   // UNI[3596] := 16#6DAE;
   // UNI[3597] := 16#6DAF;
   // UNI[3598] := 16#6DB2;
   // UNI[3599] := 16#6DB5;
   // UNI[3600] := 16#6DB8;
   // UNI[3601] := 16#6DBF;
   // UNI[3602] := 16#6DC0;
   // UNI[3603] := 16#6DC4;
   // UNI[3604] := 16#6DC5;
   // UNI[3605] := 16#6DC6;
   // UNI[3606] := 16#6DC7;
   // UNI[3607] := 16#6DCB;
   // UNI[3608] := 16#6DCC;
   // UNI[3609] := 16#6DD1;
   // UNI[3610] := 16#6DD6;
   // UNI[3611] := 16#6DD8;
   // UNI[3612] := 16#6DD9;
   // UNI[3613] := 16#6DDD;
   // UNI[3614] := 16#6DDE;
   // UNI[3615] := 16#6DE0;
   // UNI[3616] := 16#6DE1;
   // UNI[3617] := 16#6DE4;
   // UNI[3618] := 16#6DE6;
   // UNI[3619] := 16#6DEB;
   // UNI[3620] := 16#6DEC;
   // UNI[3621] := 16#6DEE;
   // UNI[3622] := 16#6DF1;
   // UNI[3623] := 16#6DF3;
   // UNI[3624] := 16#6DF7;
   // UNI[3625] := 16#6DF9;
   // UNI[3626] := 16#6DFB;
   // UNI[3627] := 16#6DFC;
   // UNI[3628] := 16#6E05;
   // UNI[3629] := 16#6E0A;
   // UNI[3630] := 16#6E0C;
   // UNI[3631] := 16#6E0D;
   // UNI[3632] := 16#6E0E;
   // UNI[3633] := 16#6E10;
   // UNI[3634] := 16#6E11;
   // UNI[3635] := 16#6E14;
   // UNI[3636] := 16#6E16;
   // UNI[3637] := 16#6E17;
   // UNI[3638] := 16#6E1A;
   // UNI[3639] := 16#6E1D;
   // UNI[3640] := 16#6E20;
   // UNI[3641] := 16#6E21;
   // UNI[3642] := 16#6E23;
   // UNI[3643] := 16#6E24;
   // UNI[3644] := 16#6E25;
   // UNI[3645] := 16#6E29;
   // UNI[3646] := 16#6E2B;
   // UNI[3647] := 16#6E2D;
   // UNI[3648] := 16#6E2F;
   // UNI[3649] := 16#6E32;
   // UNI[3650] := 16#6E34;
   // UNI[3651] := 16#6E38;
   // UNI[3652] := 16#6E3A;
   // UNI[3653] := 16#6E43;
   // UNI[3654] := 16#6E44;
   // UNI[3655] := 16#6E4D;
   // UNI[3656] := 16#6E4E;
   // UNI[3657] := 16#6E53;
   // UNI[3658] := 16#6E54;
   // UNI[3659] := 16#6E56;
   // UNI[3660] := 16#6E58;
   // UNI[3661] := 16#6E5B;
   // UNI[3662] := 16#6E5F;
   // UNI[3663] := 16#6E6B;
   // UNI[3664] := 16#6E6E;
   // UNI[3665] := 16#6E7E;
   // UNI[3666] := 16#6E7F;
   // UNI[3667] := 16#6E83;
   // UNI[3668] := 16#6E85;
   // UNI[3669] := 16#6E86;
   // UNI[3670] := 16#6E89;
   // UNI[3671] := 16#6E8F;
   // UNI[3672] := 16#6E90;
   // UNI[3673] := 16#6E98;
   // UNI[3674] := 16#6E9C;
   // UNI[3675] := 16#6E9F;
   // UNI[3676] := 16#6EA2;
   // UNI[3677] := 16#6EA5;
   // UNI[3678] := 16#6EA7;
   // UNI[3679] := 16#6EAA;
   // UNI[3680] := 16#6EAF;
   // UNI[3681] := 16#6EB1;
   // UNI[3682] := 16#6EB2;
   // UNI[3683] := 16#6EB4;
   // UNI[3684] := 16#6EB6;
   // UNI[3685] := 16#6EB7;
   // UNI[3686] := 16#6EBA;
   // UNI[3687] := 16#6EBB;
   // UNI[3688] := 16#6EBD;
   // UNI[3689] := 16#6EC1;
   // UNI[3690] := 16#6EC2;
   // UNI[3691] := 16#6EC7;
   // UNI[3692] := 16#6ECB;
   // UNI[3693] := 16#6ECF;
   // UNI[3694] := 16#6ED1;
   // UNI[3695] := 16#6ED3;
   // UNI[3696] := 16#6ED4;
   // UNI[3697] := 16#6ED5;
   // UNI[3698] := 16#6ED7;
   // UNI[3699] := 16#6EDA;
   // UNI[3700] := 16#6EDE;
   // UNI[3701] := 16#6EDF;
   // UNI[3702] := 16#6EE0;
   // UNI[3703] := 16#6EE1;
   // UNI[3704] := 16#6EE2;
   // UNI[3705] := 16#6EE4;
   // UNI[3706] := 16#6EE5;
   // UNI[3707] := 16#6EE6;
   // UNI[3708] := 16#6EE8;
   // UNI[3709] := 16#6EE9;
   // UNI[3710] := 16#6EF4;
   // UNI[3711] := 16#6EF9;
   // UNI[3712] := 16#6F02;
   // UNI[3713] := 16#6F06;
   // UNI[3714] := 16#6F09;
   // UNI[3715] := 16#6F0F;
   // UNI[3716] := 16#6F13;
   // UNI[3717] := 16#6F14;
   // UNI[3718] := 16#6F15;
   // UNI[3719] := 16#6F20;
   // UNI[3720] := 16#6F24;
   // UNI[3721] := 16#6F29;
   // UNI[3722] := 16#6F2A;
   // UNI[3723] := 16#6F2B;
   // UNI[3724] := 16#6F2D;
   // UNI[3725] := 16#6F2F;
   // UNI[3726] := 16#6F31;
   // UNI[3727] := 16#6F33;
   // UNI[3728] := 16#6F36;
   // UNI[3729] := 16#6F3E;
   // UNI[3730] := 16#6F46;
   // UNI[3731] := 16#6F47;
   // UNI[3732] := 16#6F4B;
   // UNI[3733] := 16#6F4D;
   // UNI[3734] := 16#6F58;
   // UNI[3735] := 16#6F5C;
   // UNI[3736] := 16#6F5E;
   // UNI[3737] := 16#6F62;
   // UNI[3738] := 16#6F66;
   // UNI[3739] := 16#6F6D;
   // UNI[3740] := 16#6F6E;
   // UNI[3741] := 16#6F72;
   // UNI[3742] := 16#6F74;
   // UNI[3743] := 16#6F78;
   // UNI[3744] := 16#6F7A;
   // UNI[3745] := 16#6F7C;
   // UNI[3746] := 16#6F84;
   // UNI[3747] := 16#6F88;
   // UNI[3748] := 16#6F89;
   // UNI[3749] := 16#6F8C;
   // UNI[3750] := 16#6F8D;
   // UNI[3751] := 16#6F8E;
   // UNI[3752] := 16#6F9C;
   // UNI[3753] := 16#6FA1;
   // UNI[3754] := 16#6FA7;
   // UNI[3755] := 16#6FB3;
   // UNI[3756] := 16#6FB6;
   // UNI[3757] := 16#6FB9;
   // UNI[3758] := 16#6FC0;
   // UNI[3759] := 16#6FC2;
   // UNI[3760] := 16#6FC9;
   // UNI[3761] := 16#6FD1;
   // UNI[3762] := 16#6FD2;
   // UNI[3763] := 16#6FDE;
   // UNI[3764] := 16#6FE0;
   // UNI[3765] := 16#6FE1;
   // UNI[3766] := 16#6FEE;
   // UNI[3767] := 16#6FEF;
   // UNI[3768] := 16#7011;
   // UNI[3769] := 16#701A;
   // UNI[3770] := 16#701B;
   // UNI[3771] := 16#7023;
   // UNI[3772] := 16#7035;
   // UNI[3773] := 16#7039;
   // UNI[3774] := 16#704C;
   // UNI[3775] := 16#704F;
   // UNI[3776] := 16#705E;
   // UNI[3777] := 16#706B;
   // UNI[3778] := 16#706C;
   // UNI[3779] := 16#706D;
   // UNI[3780] := 16#706F;
   // UNI[3781] := 16#7070;
   // UNI[3782] := 16#7075;
   // UNI[3783] := 16#7076;
   // UNI[3784] := 16#7078;
   // UNI[3785] := 16#707C;
   // UNI[3786] := 16#707E;
   // UNI[3787] := 16#707F;
   // UNI[3788] := 16#7080;
   // UNI[3789] := 16#7085;
   // UNI[3790] := 16#7089;
   // UNI[3791] := 16#708A;
   // UNI[3792] := 16#708E;
   // UNI[3793] := 16#7092;
   // UNI[3794] := 16#7094;
   // UNI[3795] := 16#7095;
   // UNI[3796] := 16#7096;
   // UNI[3797] := 16#7099;
   // UNI[3798] := 16#709C;
   // UNI[3799] := 16#709D;
   // UNI[3800] := 16#70AB;
   // UNI[3801] := 16#70AC;
   // UNI[3802] := 16#70AD;
   // UNI[3803] := 16#70AE;
   // UNI[3804] := 16#70AF;
   // UNI[3805] := 16#70B1;
   // UNI[3806] := 16#70B3;
   // UNI[3807] := 16#70B7;
   // UNI[3808] := 16#70B8;
   // UNI[3809] := 16#70B9;
   // UNI[3810] := 16#70BB;
   // UNI[3811] := 16#70BC;
   // UNI[3812] := 16#70BD;
   // UNI[3813] := 16#70C0;
   // UNI[3814] := 16#70C1;
   // UNI[3815] := 16#70C2;
   // UNI[3816] := 16#70C3;
   // UNI[3817] := 16#70C8;
   // UNI[3818] := 16#70CA;
   // UNI[3819] := 16#70D8;
   // UNI[3820] := 16#70D9;
   // UNI[3821] := 16#70DB;
   // UNI[3822] := 16#70DF;
   // UNI[3823] := 16#70E4;
   // UNI[3824] := 16#70E6;
   // UNI[3825] := 16#70E7;
   // UNI[3826] := 16#70E8;
   // UNI[3827] := 16#70E9;
   // UNI[3828] := 16#70EB;
   // UNI[3829] := 16#70EC;
   // UNI[3830] := 16#70ED;
   // UNI[3831] := 16#70EF;
   // UNI[3832] := 16#70F7;
   // UNI[3833] := 16#70F9;
   // UNI[3834] := 16#70FD;
   // UNI[3835] := 16#7109;
   // UNI[3836] := 16#710A;
   // UNI[3837] := 16#7110;
   // UNI[3838] := 16#7113;
   // UNI[3839] := 16#7115;
   // UNI[3840] := 16#7116;
   // UNI[3841] := 16#7118;
   // UNI[3842] := 16#7119;
   // UNI[3843] := 16#711A;
   // UNI[3844] := 16#7126;
   // UNI[3845] := 16#712F;
   // UNI[3846] := 16#7130;
   // UNI[3847] := 16#7131;
   // UNI[3848] := 16#7136;
   // UNI[3849] := 16#7145;
   // UNI[3850] := 16#714A;
   // UNI[3851] := 16#714C;
   // UNI[3852] := 16#714E;
   // UNI[3853] := 16#715C;
   // UNI[3854] := 16#715E;
   // UNI[3855] := 16#7164;
   // UNI[3856] := 16#7166;
   // UNI[3857] := 16#7167;
   // UNI[3858] := 16#7168;
   // UNI[3859] := 16#716E;
   // UNI[3860] := 16#7172;
   // UNI[3861] := 16#7173;
   // UNI[3862] := 16#7178;
   // UNI[3863] := 16#717A;
   // UNI[3864] := 16#717D;
   // UNI[3865] := 16#7184;
   // UNI[3866] := 16#718A;
   // UNI[3867] := 16#718F;
   // UNI[3868] := 16#7194;
   // UNI[3869] := 16#7198;
   // UNI[3870] := 16#7199;
   // UNI[3871] := 16#719F;
   // UNI[3872] := 16#71A0;
   // UNI[3873] := 16#71A8;
   // UNI[3874] := 16#71AC;
   // UNI[3875] := 16#71B3;
   // UNI[3876] := 16#71B5;
   // UNI[3877] := 16#71B9;
   // UNI[3878] := 16#71C3;
   // UNI[3879] := 16#71CE;
   // UNI[3880] := 16#71D4;
   // UNI[3881] := 16#71D5;
   // UNI[3882] := 16#71E0;
   // UNI[3883] := 16#71E5;
   // UNI[3884] := 16#71E7;
   // UNI[3885] := 16#71EE;
   // UNI[3886] := 16#71F9;
   // UNI[3887] := 16#7206;
   // UNI[3888] := 16#721D;
   // UNI[3889] := 16#7228;
   // UNI[3890] := 16#722A;
   // UNI[3891] := 16#722C;
   // UNI[3892] := 16#7230;
   // UNI[3893] := 16#7231;
   // UNI[3894] := 16#7235;
   // UNI[3895] := 16#7236;
   // UNI[3896] := 16#7237;
   // UNI[3897] := 16#7238;
   // UNI[3898] := 16#7239;
   // UNI[3899] := 16#723B;
   // UNI[3900] := 16#723D;
   // UNI[3901] := 16#723F;
   // UNI[3902] := 16#7247;
   // UNI[3903] := 16#7248;
   // UNI[3904] := 16#724C;
   // UNI[3905] := 16#724D;
   // UNI[3906] := 16#7252;
   // UNI[3907] := 16#7256;
   // UNI[3908] := 16#7259;
   // UNI[3909] := 16#725B;
   // UNI[3910] := 16#725D;
   // UNI[3911] := 16#725F;
   // UNI[3912] := 16#7261;
   // UNI[3913] := 16#7262;
   // UNI[3914] := 16#7266;
   // UNI[3915] := 16#7267;
   // UNI[3916] := 16#7269;
   // UNI[3917] := 16#726E;
   // UNI[3918] := 16#726F;
   // UNI[3919] := 16#7272;
   // UNI[3920] := 16#7275;
   // UNI[3921] := 16#7279;
   // UNI[3922] := 16#727A;
   // UNI[3923] := 16#727E;
   // UNI[3924] := 16#727F;
   // UNI[3925] := 16#7280;
   // UNI[3926] := 16#7281;
   // UNI[3927] := 16#7284;
   // UNI[3928] := 16#728A;
   // UNI[3929] := 16#728B;
   // UNI[3930] := 16#728D;
   // UNI[3931] := 16#728F;
   // UNI[3932] := 16#7292;
   // UNI[3933] := 16#729F;
   // UNI[3934] := 16#72AC;
   // UNI[3935] := 16#72AD;
   // UNI[3936] := 16#72AF;
   // UNI[3937] := 16#72B0;
   // UNI[3938] := 16#72B4;
   // UNI[3939] := 16#72B6;
   // UNI[3940] := 16#72B7;
   // UNI[3941] := 16#72B8;
   // UNI[3942] := 16#72B9;
   // UNI[3943] := 16#72C1;
   // UNI[3944] := 16#72C2;
   // UNI[3945] := 16#72C3;
   // UNI[3946] := 16#72C4;
   // UNI[3947] := 16#72C8;
   // UNI[3948] := 16#72CD;
   // UNI[3949] := 16#72CE;
   // UNI[3950] := 16#72D0;
   // UNI[3951] := 16#72D2;
   // UNI[3952] := 16#72D7;
   // UNI[3953] := 16#72D9;
   // UNI[3954] := 16#72DE;
   // UNI[3955] := 16#72E0;
   // UNI[3956] := 16#72E1;
   // UNI[3957] := 16#72E8;
   // UNI[3958] := 16#72E9;
   // UNI[3959] := 16#72EC;
   // UNI[3960] := 16#72ED;
   // UNI[3961] := 16#72EE;
   // UNI[3962] := 16#72EF;
   // UNI[3963] := 16#72F0;
   // UNI[3964] := 16#72F1;
   // UNI[3965] := 16#72F2;
   // UNI[3966] := 16#72F3;
   // UNI[3967] := 16#72F4;
   // UNI[3968] := 16#72F7;
   // UNI[3969] := 16#72F8;
   // UNI[3970] := 16#72FA;
   // UNI[3971] := 16#72FB;
   // UNI[3972] := 16#72FC;
   // UNI[3973] := 16#7301;
   // UNI[3974] := 16#7303;
   // UNI[3975] := 16#730A;
   // UNI[3976] := 16#730E;
   // UNI[3977] := 16#7313;
   // UNI[3978] := 16#7315;
   // UNI[3979] := 16#7316;
   // UNI[3980] := 16#7317;
   // UNI[3981] := 16#731B;
   // UNI[3982] := 16#731C;
   // UNI[3983] := 16#731D;
   // UNI[3984] := 16#731E;
   // UNI[3985] := 16#7321;
   // UNI[3986] := 16#7322;
   // UNI[3987] := 16#7325;
   // UNI[3988] := 16#7329;
   // UNI[3989] := 16#732A;
   // UNI[3990] := 16#732B;
   // UNI[3991] := 16#732C;
   // UNI[3992] := 16#732E;
   // UNI[3993] := 16#7331;
   // UNI[3994] := 16#7334;
   // UNI[3995] := 16#7337;
   // UNI[3996] := 16#7338;
   // UNI[3997] := 16#7339;
   // UNI[3998] := 16#733E;
   // UNI[3999] := 16#733F;
   // UNI[4000] := 16#734D;
   // UNI[4001] := 16#7350;
   // UNI[4002] := 16#7352;
   // UNI[4003] := 16#7357;
   // UNI[4004] := 16#7360;
   // UNI[4005] := 16#736C;
   // UNI[4006] := 16#736D;
   // UNI[4007] := 16#736F;
   // UNI[4008] := 16#737E;
   // UNI[4009] := 16#7384;
   // UNI[4010] := 16#7387;
   // UNI[4011] := 16#7389;
   // UNI[4012] := 16#738B;
   // UNI[4013] := 16#738E;
   // UNI[4014] := 16#7391;
   // UNI[4015] := 16#7396;
   // UNI[4016] := 16#739B;
   // UNI[4017] := 16#739F;
   // UNI[4018] := 16#73A2;
   // UNI[4019] := 16#73A9;
   // UNI[4020] := 16#73AB;
   // UNI[4021] := 16#73AE;
   // UNI[4022] := 16#73AF;
   // UNI[4023] := 16#73B0;
   // UNI[4024] := 16#73B2;
   // UNI[4025] := 16#73B3;
   // UNI[4026] := 16#73B7;
   // UNI[4027] := 16#73BA;
   // UNI[4028] := 16#73BB;
   // UNI[4029] := 16#73C0;
   // UNI[4030] := 16#73C2;
   // UNI[4031] := 16#73C8;
   // UNI[4032] := 16#73C9;
   // UNI[4033] := 16#73CA;
   // UNI[4034] := 16#73CD;
   // UNI[4035] := 16#73CF;
   // UNI[4036] := 16#73D0;
   // UNI[4037] := 16#73D1;
   // UNI[4038] := 16#73D9;
   // UNI[4039] := 16#73DE;
   // UNI[4040] := 16#73E0;
   // UNI[4041] := 16#73E5;
   // UNI[4042] := 16#73E7;
   // UNI[4043] := 16#73E9;
   // UNI[4044] := 16#73ED;
   // UNI[4045] := 16#73F2;
   // UNI[4046] := 16#7403;
   // UNI[4047] := 16#7405;
   // UNI[4048] := 16#7406;
   // UNI[4049] := 16#7409;
   // UNI[4050] := 16#740A;
   // UNI[4051] := 16#740F;
   // UNI[4052] := 16#7410;
   // UNI[4053] := 16#741A;
   // UNI[4054] := 16#741B;
   // UNI[4055] := 16#7422;
   // UNI[4056] := 16#7425;
   // UNI[4057] := 16#7426;
   // UNI[4058] := 16#7428;
   // UNI[4059] := 16#742A;
   // UNI[4060] := 16#742C;
   // UNI[4061] := 16#742E;
   // UNI[4062] := 16#7430;
   // UNI[4063] := 16#7433;
   // UNI[4064] := 16#7434;
   // UNI[4065] := 16#7435;
   // UNI[4066] := 16#7436;
   // UNI[4067] := 16#743C;
   // UNI[4068] := 16#7441;
   // UNI[4069] := 16#7455;
   // UNI[4070] := 16#7457;
   // UNI[4071] := 16#7459;
   // UNI[4072] := 16#745A;
   // UNI[4073] := 16#745B;
   // UNI[4074] := 16#745C;
   // UNI[4075] := 16#745E;
   // UNI[4076] := 16#745F;
   // UNI[4077] := 16#746D;
   // UNI[4078] := 16#7470;
   // UNI[4079] := 16#7476;
   // UNI[4080] := 16#7477;
   // UNI[4081] := 16#747E;
   // UNI[4082] := 16#7480;
   // UNI[4083] := 16#7481;
   // UNI[4084] := 16#7483;
   // UNI[4085] := 16#7487;
   // UNI[4086] := 16#748B;
   // UNI[4087] := 16#748E;
   // UNI[4088] := 16#7490;
   // UNI[4089] := 16#749C;
   // UNI[4090] := 16#749E;
   // UNI[4091] := 16#74A7;
   // UNI[4092] := 16#74A8;
   // UNI[4093] := 16#74A9;
   // UNI[4094] := 16#74BA;
   // UNI[4095] := 16#74D2;
   // UNI[4096] := 16#74DC;
   // UNI[4097] := 16#74DE;
   // UNI[4098] := 16#74E0;
   // UNI[4099] := 16#74E2;
   // UNI[4100] := 16#74E3;
   // UNI[4101] := 16#74E4;
   // UNI[4102] := 16#74E6;
   // UNI[4103] := 16#74EE;
   // UNI[4104] := 16#74EF;
   // UNI[4105] := 16#74F4;
   // UNI[4106] := 16#74F6;
   // UNI[4107] := 16#74F7;
   // UNI[4108] := 16#74FF;
   // UNI[4109] := 16#7504;
   // UNI[4110] := 16#750D;
   // UNI[4111] := 16#750F;
   // UNI[4112] := 16#7511;
   // UNI[4113] := 16#7513;
   // UNI[4114] := 16#7518;
   // UNI[4115] := 16#7519;
   // UNI[4116] := 16#751A;
   // UNI[4117] := 16#751C;
   // UNI[4118] := 16#751F;
   // UNI[4119] := 16#7525;
   // UNI[4120] := 16#7528;
   // UNI[4121] := 16#7529;
   // UNI[4122] := 16#752B;
   // UNI[4123] := 16#752C;
   // UNI[4124] := 16#752D;
   // UNI[4125] := 16#752F;
   // UNI[4126] := 16#7530;
   // UNI[4127] := 16#7531;
   // UNI[4128] := 16#7532;
   // UNI[4129] := 16#7533;
   // UNI[4130] := 16#7535;
   // UNI[4131] := 16#7537;
   // UNI[4132] := 16#7538;
   // UNI[4133] := 16#753A;
   // UNI[4134] := 16#753B;
   // UNI[4135] := 16#753E;
   // UNI[4136] := 16#7540;
   // UNI[4137] := 16#7545;
   // UNI[4138] := 16#7548;
   // UNI[4139] := 16#754B;
   // UNI[4140] := 16#754C;
   // UNI[4141] := 16#754E;
   // UNI[4142] := 16#754F;
   // UNI[4143] := 16#7554;
   // UNI[4144] := 16#7559;
   // UNI[4145] := 16#755A;
   // UNI[4146] := 16#755B;
   // UNI[4147] := 16#755C;
   // UNI[4148] := 16#7565;
   // UNI[4149] := 16#7566;
   // UNI[4150] := 16#756A;
   // UNI[4151] := 16#7572;
   // UNI[4152] := 16#7574;
   // UNI[4153] := 16#7578;
   // UNI[4154] := 16#7579;
   // UNI[4155] := 16#757F;
   // UNI[4156] := 16#7583;
   // UNI[4157] := 16#7586;
   // UNI[4158] := 16#758B;
   // UNI[4159] := 16#758F;
   // UNI[4160] := 16#7591;
   // UNI[4161] := 16#7592;
   // UNI[4162] := 16#7594;
   // UNI[4163] := 16#7596;
   // UNI[4164] := 16#7597;
   // UNI[4165] := 16#7599;
   // UNI[4166] := 16#759A;
   // UNI[4167] := 16#759D;
   // UNI[4168] := 16#759F;
   // UNI[4169] := 16#75A0;
   // UNI[4170] := 16#75A1;
   // UNI[4171] := 16#75A3;
   // UNI[4172] := 16#75A4;
   // UNI[4173] := 16#75A5;
   // UNI[4174] := 16#75AB;
   // UNI[4175] := 16#75AC;
   // UNI[4176] := 16#75AE;
   // UNI[4177] := 16#75AF;
   // UNI[4178] := 16#75B0;
   // UNI[4179] := 16#75B1;
   // UNI[4180] := 16#75B2;
   // UNI[4181] := 16#75B3;
   // UNI[4182] := 16#75B4;
   // UNI[4183] := 16#75B5;
   // UNI[4184] := 16#75B8;
   // UNI[4185] := 16#75B9;
   // UNI[4186] := 16#75BC;
   // UNI[4187] := 16#75BD;
   // UNI[4188] := 16#75BE;
   // UNI[4189] := 16#75C2;
   // UNI[4190] := 16#75C3;
   // UNI[4191] := 16#75C4;
   // UNI[4192] := 16#75C5;
   // UNI[4193] := 16#75C7;
   // UNI[4194] := 16#75C8;
   // UNI[4195] := 16#75C9;
   // UNI[4196] := 16#75CA;
   // UNI[4197] := 16#75CD;
   // UNI[4198] := 16#75D2;
   // UNI[4199] := 16#75D4;
   // UNI[4200] := 16#75D5;
   // UNI[4201] := 16#75D6;
   // UNI[4202] := 16#75D8;
   // UNI[4203] := 16#75DB;
   // UNI[4204] := 16#75DE;
   // UNI[4205] := 16#75E2;
   // UNI[4206] := 16#75E3;
   // UNI[4207] := 16#75E4;
   // UNI[4208] := 16#75E6;
   // UNI[4209] := 16#75E7;
   // UNI[4210] := 16#75E8;
   // UNI[4211] := 16#75EA;
   // UNI[4212] := 16#75EB;
   // UNI[4213] := 16#75F0;
   // UNI[4214] := 16#75F1;
   // UNI[4215] := 16#75F4;
   // UNI[4216] := 16#75F9;
   // UNI[4217] := 16#75FC;
   // UNI[4218] := 16#75FF;
   // UNI[4219] := 16#7600;
   // UNI[4220] := 16#7601;
   // UNI[4221] := 16#7603;
   // UNI[4222] := 16#7605;
   // UNI[4223] := 16#760A;
   // UNI[4224] := 16#760C;
   // UNI[4225] := 16#7610;
   // UNI[4226] := 16#7615;
   // UNI[4227] := 16#7617;
   // UNI[4228] := 16#7618;
   // UNI[4229] := 16#7619;
   // UNI[4230] := 16#761B;
   // UNI[4231] := 16#761F;
   // UNI[4232] := 16#7620;
   // UNI[4233] := 16#7622;
   // UNI[4234] := 16#7624;
   // UNI[4235] := 16#7625;
   // UNI[4236] := 16#7626;
   // UNI[4237] := 16#7629;
   // UNI[4238] := 16#762A;
   // UNI[4239] := 16#762B;
   // UNI[4240] := 16#762D;
   // UNI[4241] := 16#7630;
   // UNI[4242] := 16#7633;
   // UNI[4243] := 16#7634;
   // UNI[4244] := 16#7635;
   // UNI[4245] := 16#7638;
   // UNI[4246] := 16#763C;
   // UNI[4247] := 16#763E;
   // UNI[4248] := 16#763F;
   // UNI[4249] := 16#7640;
   // UNI[4250] := 16#7643;
   // UNI[4251] := 16#764C;
   // UNI[4252] := 16#764D;
   // UNI[4253] := 16#7654;
   // UNI[4254] := 16#7656;
   // UNI[4255] := 16#765C;
   // UNI[4256] := 16#765E;
   // UNI[4257] := 16#7663;
   // UNI[4258] := 16#766B;
   // UNI[4259] := 16#766F;
   // UNI[4260] := 16#7678;
   // UNI[4261] := 16#767B;
   // UNI[4262] := 16#767D;
   // UNI[4263] := 16#767E;
   // UNI[4264] := 16#7682;
   // UNI[4265] := 16#7684;
   // UNI[4266] := 16#7686;
   // UNI[4267] := 16#7687;
   // UNI[4268] := 16#7688;
   // UNI[4269] := 16#768B;
   // UNI[4270] := 16#768E;
   // UNI[4271] := 16#7691;
   // UNI[4272] := 16#7693;
   // UNI[4273] := 16#7696;
   // UNI[4274] := 16#7699;
   // UNI[4275] := 16#76A4;
   // UNI[4276] := 16#76AE;
   // UNI[4277] := 16#76B1;
   // UNI[4278] := 16#76B2;
   // UNI[4279] := 16#76B4;
   // UNI[4280] := 16#76BF;
   // UNI[4281] := 16#76C2;
   // UNI[4282] := 16#76C5;
   // UNI[4283] := 16#76C6;
   // UNI[4284] := 16#76C8;
   // UNI[4285] := 16#76CA;
   // UNI[4286] := 16#76CD;
   // UNI[4287] := 16#76CE;
   // UNI[4288] := 16#76CF;
   // UNI[4289] := 16#76D0;
   // UNI[4290] := 16#76D1;
   // UNI[4291] := 16#76D2;
   // UNI[4292] := 16#76D4;
   // UNI[4293] := 16#76D6;
   // UNI[4294] := 16#76D7;
   // UNI[4295] := 16#76D8;
   // UNI[4296] := 16#76DB;
   // UNI[4297] := 16#76DF;
   // UNI[4298] := 16#76E5;
   // UNI[4299] := 16#76EE;
   // UNI[4300] := 16#76EF;
   // UNI[4301] := 16#76F1;
   // UNI[4302] := 16#76F2;
   // UNI[4303] := 16#76F4;
   // UNI[4304] := 16#76F8;
   // UNI[4305] := 16#76F9;
   // UNI[4306] := 16#76FC;
   // UNI[4307] := 16#76FE;
   // UNI[4308] := 16#7701;
   // UNI[4309] := 16#7704;
   // UNI[4310] := 16#7707;
   // UNI[4311] := 16#7708;
   // UNI[4312] := 16#7709;
   // UNI[4313] := 16#770B;
   // UNI[4314] := 16#770D;
   // UNI[4315] := 16#7719;
   // UNI[4316] := 16#771A;
   // UNI[4317] := 16#771F;
   // UNI[4318] := 16#7720;
   // UNI[4319] := 16#7722;
   // UNI[4320] := 16#7726;
   // UNI[4321] := 16#7728;
   // UNI[4322] := 16#7729;
   // UNI[4323] := 16#772D;
   // UNI[4324] := 16#772F;
   // UNI[4325] := 16#7735;
   // UNI[4326] := 16#7736;
   // UNI[4327] := 16#7737;
   // UNI[4328] := 16#7738;
   // UNI[4329] := 16#773A;
   // UNI[4330] := 16#773C;
   // UNI[4331] := 16#7740;
   // UNI[4332] := 16#7741;
   // UNI[4333] := 16#7743;
   // UNI[4334] := 16#7747;
   // UNI[4335] := 16#7750;
   // UNI[4336] := 16#7751;
   // UNI[4337] := 16#775A;
   // UNI[4338] := 16#775B;
   // UNI[4339] := 16#7761;
   // UNI[4340] := 16#7762;
   // UNI[4341] := 16#7763;
   // UNI[4342] := 16#7765;
   // UNI[4343] := 16#7766;
   // UNI[4344] := 16#7768;
   // UNI[4345] := 16#776B;
   // UNI[4346] := 16#776C;
   // UNI[4347] := 16#7779;
   // UNI[4348] := 16#777D;
   // UNI[4349] := 16#777E;
   // UNI[4350] := 16#777F;
   // UNI[4351] := 16#7780;
   // UNI[4352] := 16#7784;
   // UNI[4353] := 16#7785;
   // UNI[4354] := 16#778C;
   // UNI[4355] := 16#778D;
   // UNI[4356] := 16#778E;
   // UNI[4357] := 16#7791;
   // UNI[4358] := 16#7792;
   // UNI[4359] := 16#779F;
   // UNI[4360] := 16#77A0;
   // UNI[4361] := 16#77A2;
   // UNI[4362] := 16#77A5;
   // UNI[4363] := 16#77A7;
   // UNI[4364] := 16#77A9;
   // UNI[4365] := 16#77AA;
   // UNI[4366] := 16#77AC;
   // UNI[4367] := 16#77B0;
   // UNI[4368] := 16#77B3;
   // UNI[4369] := 16#77B5;
   // UNI[4370] := 16#77BB;
   // UNI[4371] := 16#77BD;
   // UNI[4372] := 16#77BF;
   // UNI[4373] := 16#77CD;
   // UNI[4374] := 16#77D7;
   // UNI[4375] := 16#77DB;
   // UNI[4376] := 16#77DC;
   // UNI[4377] := 16#77E2;
   // UNI[4378] := 16#77E3;
   // UNI[4379] := 16#77E5;
   // UNI[4380] := 16#77E7;
   // UNI[4381] := 16#77E9;
   // UNI[4382] := 16#77EB;
   // UNI[4383] := 16#77EC;
   // UNI[4384] := 16#77ED;
   // UNI[4385] := 16#77EE;
   // UNI[4386] := 16#77F3;
   // UNI[4387] := 16#77F6;
   // UNI[4388] := 16#77F8;
   // UNI[4389] := 16#77FD;
   // UNI[4390] := 16#77FE;
   // UNI[4391] := 16#77FF;
   // UNI[4392] := 16#7800;
   // UNI[4393] := 16#7801;
   // UNI[4394] := 16#7802;
   // UNI[4395] := 16#7809;
   // UNI[4396] := 16#780C;
   // UNI[4397] := 16#780D;
   // UNI[4398] := 16#7811;
   // UNI[4399] := 16#7812;
   // UNI[4400] := 16#7814;
   // UNI[4401] := 16#7816;
   // UNI[4402] := 16#7817;
   // UNI[4403] := 16#7818;
   // UNI[4404] := 16#781A;
   // UNI[4405] := 16#781C;
   // UNI[4406] := 16#781D;
   // UNI[4407] := 16#781F;
   // UNI[4408] := 16#7823;
   // UNI[4409] := 16#7825;
   // UNI[4410] := 16#7826;
   // UNI[4411] := 16#7827;
   // UNI[4412] := 16#7829;
   // UNI[4413] := 16#782C;
   // UNI[4414] := 16#782D;
   // UNI[4415] := 16#7830;
   // UNI[4416] := 16#7834;
   // UNI[4417] := 16#7837;
   // UNI[4418] := 16#7838;
   // UNI[4419] := 16#7839;
   // UNI[4420] := 16#783A;
   // UNI[4421] := 16#783B;
   // UNI[4422] := 16#783C;
   // UNI[4423] := 16#783E;
   // UNI[4424] := 16#7840;
   // UNI[4425] := 16#7845;
   // UNI[4426] := 16#7847;
   // UNI[4427] := 16#784C;
   // UNI[4428] := 16#784E;
   // UNI[4429] := 16#7850;
   // UNI[4430] := 16#7852;
   // UNI[4431] := 16#7855;
   // UNI[4432] := 16#7856;
   // UNI[4433] := 16#7857;
   // UNI[4434] := 16#785D;
   // UNI[4435] := 16#786A;
   // UNI[4436] := 16#786B;
   // UNI[4437] := 16#786C;
   // UNI[4438] := 16#786D;
   // UNI[4439] := 16#786E;
   // UNI[4440] := 16#7877;
   // UNI[4441] := 16#787C;
   // UNI[4442] := 16#7887;
   // UNI[4443] := 16#7889;
   // UNI[4444] := 16#788C;
   // UNI[4445] := 16#788D;
   // UNI[4446] := 16#788E;
   // UNI[4447] := 16#7891;
   // UNI[4448] := 16#7893;
   // UNI[4449] := 16#7897;
   // UNI[4450] := 16#7898;
   // UNI[4451] := 16#789A;
   // UNI[4452] := 16#789B;
   // UNI[4453] := 16#789C;
   // UNI[4454] := 16#789F;
   // UNI[4455] := 16#78A1;
   // UNI[4456] := 16#78A3;
   // UNI[4457] := 16#78A5;
   // UNI[4458] := 16#78A7;
   // UNI[4459] := 16#78B0;
   // UNI[4460] := 16#78B1;
   // UNI[4461] := 16#78B2;
   // UNI[4462] := 16#78B3;
   // UNI[4463] := 16#78B4;
   // UNI[4464] := 16#78B9;
   // UNI[4465] := 16#78BE;
   // UNI[4466] := 16#78C1;
   // UNI[4467] := 16#78C5;
   // UNI[4468] := 16#78C9;
   // UNI[4469] := 16#78CA;
   // UNI[4470] := 16#78CB;
   // UNI[4471] := 16#78D0;
   // UNI[4472] := 16#78D4;
   // UNI[4473] := 16#78D5;
   // UNI[4474] := 16#78D9;
   // UNI[4475] := 16#78E8;
   // UNI[4476] := 16#78EC;
   // UNI[4477] := 16#78F2;
   // UNI[4478] := 16#78F4;
   // UNI[4479] := 16#78F7;
   // UNI[4480] := 16#78FA;
   // UNI[4481] := 16#7901;
   // UNI[4482] := 16#7905;
   // UNI[4483] := 16#7913;
   // UNI[4484] := 16#791E;
   // UNI[4485] := 16#7924;
   // UNI[4486] := 16#7934;
   // UNI[4487] := 16#793A;
   // UNI[4488] := 16#793B;
   // UNI[4489] := 16#793C;
   // UNI[4490] := 16#793E;
   // UNI[4491] := 16#7940;
   // UNI[4492] := 16#7941;
   // UNI[4493] := 16#7946;
   // UNI[4494] := 16#7948;
   // UNI[4495] := 16#7949;
   // UNI[4496] := 16#7953;
   // UNI[4497] := 16#7956;
   // UNI[4498] := 16#7957;
   // UNI[4499] := 16#795A;
   // UNI[4500] := 16#795B;
   // UNI[4501] := 16#795C;
   // UNI[4502] := 16#795D;
   // UNI[4503] := 16#795E;
   // UNI[4504] := 16#795F;
   // UNI[4505] := 16#7960;
   // UNI[4506] := 16#7962;
   // UNI[4507] := 16#7965;
   // UNI[4508] := 16#7967;
   // UNI[4509] := 16#7968;
   // UNI[4510] := 16#796D;
   // UNI[4511] := 16#796F;
   // UNI[4512] := 16#7977;
   // UNI[4513] := 16#7978;
   // UNI[4514] := 16#797A;
   // UNI[4515] := 16#7980;
   // UNI[4516] := 16#7981;
   // UNI[4517] := 16#7984;
   // UNI[4518] := 16#7985;
   // UNI[4519] := 16#798A;
   // UNI[4520] := 16#798F;
   // UNI[4521] := 16#799A;
   // UNI[4522] := 16#79A7;
   // UNI[4523] := 16#79B3;
   // UNI[4524] := 16#79B9;
   // UNI[4525] := 16#79BA;
   // UNI[4526] := 16#79BB;
   // UNI[4527] := 16#79BD;
   // UNI[4528] := 16#79BE;
   // UNI[4529] := 16#79C0;
   // UNI[4530] := 16#79C1;
   // UNI[4531] := 16#79C3;
   // UNI[4532] := 16#79C6;
   // UNI[4533] := 16#79C9;
   // UNI[4534] := 16#79CB;
   // UNI[4535] := 16#79CD;
   // UNI[4536] := 16#79D1;
   // UNI[4537] := 16#79D2;
   // UNI[4538] := 16#79D5;
   // UNI[4539] := 16#79D8;
   // UNI[4540] := 16#79DF;
   // UNI[4541] := 16#79E3;
   // UNI[4542] := 16#79E4;
   // UNI[4543] := 16#79E6;
   // UNI[4544] := 16#79E7;
   // UNI[4545] := 16#79E9;
   // UNI[4546] := 16#79EB;
   // UNI[4547] := 16#79ED;
   // UNI[4548] := 16#79EF;
   // UNI[4549] := 16#79F0;
   // UNI[4550] := 16#79F8;
   // UNI[4551] := 16#79FB;
   // UNI[4552] := 16#79FD;
   // UNI[4553] := 16#7A00;
   // UNI[4554] := 16#7A02;
   // UNI[4555] := 16#7A03;
   // UNI[4556] := 16#7A06;
   // UNI[4557] := 16#7A0B;
   // UNI[4558] := 16#7A0D;
   // UNI[4559] := 16#7A0E;
   // UNI[4560] := 16#7A14;
   // UNI[4561] := 16#7A17;
   // UNI[4562] := 16#7A1A;
   // UNI[4563] := 16#7A1E;
   // UNI[4564] := 16#7A20;
   // UNI[4565] := 16#7A23;
   // UNI[4566] := 16#7A33;
   // UNI[4567] := 16#7A37;
   // UNI[4568] := 16#7A39;
   // UNI[4569] := 16#7A3B;
   // UNI[4570] := 16#7A3C;
   // UNI[4571] := 16#7A3D;
   // UNI[4572] := 16#7A3F;
   // UNI[4573] := 16#7A46;
   // UNI[4574] := 16#7A51;
   // UNI[4575] := 16#7A57;
   // UNI[4576] := 16#7A70;
   // UNI[4577] := 16#7A74;
   // UNI[4578] := 16#7A76;
   // UNI[4579] := 16#7A77;
   // UNI[4580] := 16#7A78;
   // UNI[4581] := 16#7A79;
   // UNI[4582] := 16#7A7A;
   // UNI[4583] := 16#7A7F;
   // UNI[4584] := 16#7A80;
   // UNI[4585] := 16#7A81;
   // UNI[4586] := 16#7A83;
   // UNI[4587] := 16#7A84;
   // UNI[4588] := 16#7A86;
   // UNI[4589] := 16#7A88;
   // UNI[4590] := 16#7A8D;
   // UNI[4591] := 16#7A91;
   // UNI[4592] := 16#7A92;
   // UNI[4593] := 16#7A95;
   // UNI[4594] := 16#7A96;
   // UNI[4595] := 16#7A97;
   // UNI[4596] := 16#7A98;
   // UNI[4597] := 16#7A9C;
   // UNI[4598] := 16#7A9D;
   // UNI[4599] := 16#7A9F;
   // UNI[4600] := 16#7AA0;
   // UNI[4601] := 16#7AA5;
   // UNI[4602] := 16#7AA6;
   // UNI[4603] := 16#7AA8;
   // UNI[4604] := 16#7AAC;
   // UNI[4605] := 16#7AAD;
   // UNI[4606] := 16#7AB3;
   // UNI[4607] := 16#7ABF;
   // UNI[4608] := 16#7ACB;
   // UNI[4609] := 16#7AD6;
   // UNI[4610] := 16#7AD9;
   // UNI[4611] := 16#7ADE;
   // UNI[4612] := 16#7ADF;
   // UNI[4613] := 16#7AE0;
   // UNI[4614] := 16#7AE3;
   // UNI[4615] := 16#7AE5;
   // UNI[4616] := 16#7AE6;
   // UNI[4617] := 16#7AED;
   // UNI[4618] := 16#7AEF;
   // UNI[4619] := 16#7AF9;
   // UNI[4620] := 16#7AFA;
   // UNI[4621] := 16#7AFD;
   // UNI[4622] := 16#7AFF;
   // UNI[4623] := 16#7B03;
   // UNI[4624] := 16#7B04;
   // UNI[4625] := 16#7B06;
   // UNI[4626] := 16#7B08;
   // UNI[4627] := 16#7B0A;
   // UNI[4628] := 16#7B0B;
   // UNI[4629] := 16#7B0F;
   // UNI[4630] := 16#7B11;
   // UNI[4631] := 16#7B14;
   // UNI[4632] := 16#7B15;
   // UNI[4633] := 16#7B19;
   // UNI[4634] := 16#7B1B;
   // UNI[4635] := 16#7B1E;
   // UNI[4636] := 16#7B20;
   // UNI[4637] := 16#7B24;
   // UNI[4638] := 16#7B25;
   // UNI[4639] := 16#7B26;
   // UNI[4640] := 16#7B28;
   // UNI[4641] := 16#7B2A;
   // UNI[4642] := 16#7B2B;
   // UNI[4643] := 16#7B2C;
   // UNI[4644] := 16#7B2E;
   // UNI[4645] := 16#7B31;
   // UNI[4646] := 16#7B33;
   // UNI[4647] := 16#7B38;
   // UNI[4648] := 16#7B3A;
   // UNI[4649] := 16#7B3C;
   // UNI[4650] := 16#7B3E;
   // UNI[4651] := 16#7B45;
   // UNI[4652] := 16#7B47;
   // UNI[4653] := 16#7B49;
   // UNI[4654] := 16#7B4B;
   // UNI[4655] := 16#7B4C;
   // UNI[4656] := 16#7B4F;
   // UNI[4657] := 16#7B50;
   // UNI[4658] := 16#7B51;
   // UNI[4659] := 16#7B52;
   // UNI[4660] := 16#7B54;
   // UNI[4661] := 16#7B56;
   // UNI[4662] := 16#7B58;
   // UNI[4663] := 16#7B5A;
   // UNI[4664] := 16#7B5B;
   // UNI[4665] := 16#7B5D;
   // UNI[4666] := 16#7B60;
   // UNI[4667] := 16#7B62;
   // UNI[4668] := 16#7B6E;
   // UNI[4669] := 16#7B71;
   // UNI[4670] := 16#7B72;
   // UNI[4671] := 16#7B75;
   // UNI[4672] := 16#7B77;
   // UNI[4673] := 16#7B79;
   // UNI[4674] := 16#7B7B;
   // UNI[4675] := 16#7B7E;
   // UNI[4676] := 16#7B80;
   // UNI[4677] := 16#7B85;
   // UNI[4678] := 16#7B8D;
   // UNI[4679] := 16#7B90;
   // UNI[4680] := 16#7B94;
   // UNI[4681] := 16#7B95;
   // UNI[4682] := 16#7B97;
   // UNI[4683] := 16#7B9C;
   // UNI[4684] := 16#7B9D;
   // UNI[4685] := 16#7BA1;
   // UNI[4686] := 16#7BA2;
   // UNI[4687] := 16#7BA6;
   // UNI[4688] := 16#7BA7;
   // UNI[4689] := 16#7BA8;
   // UNI[4690] := 16#7BA9;
   // UNI[4691] := 16#7BAA;
   // UNI[4692] := 16#7BAB;
   // UNI[4693] := 16#7BAC;
   // UNI[4694] := 16#7BAD;
   // UNI[4695] := 16#7BB1;
   // UNI[4696] := 16#7BB4;
   // UNI[4697] := 16#7BB8;
   // UNI[4698] := 16#7BC1;
   // UNI[4699] := 16#7BC6;
   // UNI[4700] := 16#7BC7;
   // UNI[4701] := 16#7BCC;
   // UNI[4702] := 16#7BD1;
   // UNI[4703] := 16#7BD3;
   // UNI[4704] := 16#7BD9;
   // UNI[4705] := 16#7BDA;
   // UNI[4706] := 16#7BDD;
   // UNI[4707] := 16#7BE1;
   // UNI[4708] := 16#7BE5;
   // UNI[4709] := 16#7BE6;
   // UNI[4710] := 16#7BEA;
   // UNI[4711] := 16#7BEE;
   // UNI[4712] := 16#7BF1;
   // UNI[4713] := 16#7BF7;
   // UNI[4714] := 16#7BFC;
   // UNI[4715] := 16#7BFE;
   // UNI[4716] := 16#7C07;
   // UNI[4717] := 16#7C0B;
   // UNI[4718] := 16#7C0C;
   // UNI[4719] := 16#7C0F;
   // UNI[4720] := 16#7C16;
   // UNI[4721] := 16#7C1F;
   // UNI[4722] := 16#7C26;
   // UNI[4723] := 16#7C27;
   // UNI[4724] := 16#7C2A;
   // UNI[4725] := 16#7C38;
   // UNI[4726] := 16#7C3F;
   // UNI[4727] := 16#7C40;
   // UNI[4728] := 16#7C41;
   // UNI[4729] := 16#7C4D;
   // UNI[4730] := 16#7C73;
   // UNI[4731] := 16#7C74;
   // UNI[4732] := 16#7C7B;
   // UNI[4733] := 16#7C7C;
   // UNI[4734] := 16#7C7D;
   // UNI[4735] := 16#7C89;
   // UNI[4736] := 16#7C91;
   // UNI[4737] := 16#7C92;
   // UNI[4738] := 16#7C95;
   // UNI[4739] := 16#7C97;
   // UNI[4740] := 16#7C98;
   // UNI[4741] := 16#7C9C;
   // UNI[4742] := 16#7C9D;
   // UNI[4743] := 16#7C9E;
   // UNI[4744] := 16#7C9F;
   // UNI[4745] := 16#7CA2;
   // UNI[4746] := 16#7CA4;
   // UNI[4747] := 16#7CA5;
   // UNI[4748] := 16#7CAA;
   // UNI[4749] := 16#7CAE;
   // UNI[4750] := 16#7CB1;
   // UNI[4751] := 16#7CB2;
   // UNI[4752] := 16#7CB3;
   // UNI[4753] := 16#7CB9;
   // UNI[4754] := 16#7CBC;
   // UNI[4755] := 16#7CBD;
   // UNI[4756] := 16#7CBE;
   // UNI[4757] := 16#7CC1;
   // UNI[4758] := 16#7CC5;
   // UNI[4759] := 16#7CC7;
   // UNI[4760] := 16#7CC8;
   // UNI[4761] := 16#7CCA;
   // UNI[4762] := 16#7CCC;
   // UNI[4763] := 16#7CCD;
   // UNI[4764] := 16#7CD5;
   // UNI[4765] := 16#7CD6;
   // UNI[4766] := 16#7CD7;
   // UNI[4767] := 16#7CD9;
   // UNI[4768] := 16#7CDC;
   // UNI[4769] := 16#7CDF;
   // UNI[4770] := 16#7CE0;
   // UNI[4771] := 16#7CE8;
   // UNI[4772] := 16#7CEF;
   // UNI[4773] := 16#7CF8;
   // UNI[4774] := 16#7CFB;
   // UNI[4775] := 16#7D0A;
   // UNI[4776] := 16#7D20;
   // UNI[4777] := 16#7D22;
   // UNI[4778] := 16#7D27;
   // UNI[4779] := 16#7D2B;
   // UNI[4780] := 16#7D2F;
   // UNI[4781] := 16#7D6E;
   // UNI[4782] := 16#7D77;
   // UNI[4783] := 16#7DA6;
   // UNI[4784] := 16#7DAE;
   // UNI[4785] := 16#7E3B;
   // UNI[4786] := 16#7E41;
   // UNI[4787] := 16#7E47;
   // UNI[4788] := 16#7E82;
   // UNI[4789] := 16#7E9B;
   // UNI[4790] := 16#7E9F;
   // UNI[4791] := 16#7EA0;
   // UNI[4792] := 16#7EA1;
   // UNI[4793] := 16#7EA2;
   // UNI[4794] := 16#7EA3;
   // UNI[4795] := 16#7EA4;
   // UNI[4796] := 16#7EA5;
   // UNI[4797] := 16#7EA6;
   // UNI[4798] := 16#7EA7;
   // UNI[4799] := 16#7EA8;
   // UNI[4800] := 16#7EA9;
   // UNI[4801] := 16#7EAA;
   // UNI[4802] := 16#7EAB;
   // UNI[4803] := 16#7EAC;
   // UNI[4804] := 16#7EAD;
   // UNI[4805] := 16#7EAF;
   // UNI[4806] := 16#7EB0;
   // UNI[4807] := 16#7EB1;
   // UNI[4808] := 16#7EB2;
   // UNI[4809] := 16#7EB3;
   // UNI[4810] := 16#7EB5;
   // UNI[4811] := 16#7EB6;
   // UNI[4812] := 16#7EB7;
   // UNI[4813] := 16#7EB8;
   // UNI[4814] := 16#7EB9;
   // UNI[4815] := 16#7EBA;
   // UNI[4816] := 16#7EBD;
   // UNI[4817] := 16#7EBE;
   // UNI[4818] := 16#7EBF;
   // UNI[4819] := 16#7EC0;
   // UNI[4820] := 16#7EC1;
   // UNI[4821] := 16#7EC2;
   // UNI[4822] := 16#7EC3;
   // UNI[4823] := 16#7EC4;
   // UNI[4824] := 16#7EC5;
   // UNI[4825] := 16#7EC6;
   // UNI[4826] := 16#7EC7;
   // UNI[4827] := 16#7EC8;
   // UNI[4828] := 16#7EC9;
   // UNI[4829] := 16#7ECA;
   // UNI[4830] := 16#7ECB;
   // UNI[4831] := 16#7ECC;
   // UNI[4832] := 16#7ECD;
   // UNI[4833] := 16#7ECE;
   // UNI[4834] := 16#7ECF;
   // UNI[4835] := 16#7ED0;
   // UNI[4836] := 16#7ED1;
   // UNI[4837] := 16#7ED2;
   // UNI[4838] := 16#7ED3;
   // UNI[4839] := 16#7ED4;
   // UNI[4840] := 16#7ED5;
   // UNI[4841] := 16#7ED7;
   // UNI[4842] := 16#7ED8;
   // UNI[4843] := 16#7ED9;
   // UNI[4844] := 16#7EDA;
   // UNI[4845] := 16#7EDB;
   // UNI[4846] := 16#7EDC;
   // UNI[4847] := 16#7EDD;
   // UNI[4848] := 16#7EDE;
   // UNI[4849] := 16#7EDF;
   // UNI[4850] := 16#7EE0;
   // UNI[4851] := 16#7EE1;
   // UNI[4852] := 16#7EE2;
   // UNI[4853] := 16#7EE3;
   // UNI[4854] := 16#7EE5;
   // UNI[4855] := 16#7EE6;
   // UNI[4856] := 16#7EE7;
   // UNI[4857] := 16#7EE8;
   // UNI[4858] := 16#7EE9;
   // UNI[4859] := 16#7EEA;
   // UNI[4860] := 16#7EEB;
   // UNI[4861] := 16#7EED;
   // UNI[4862] := 16#7EEE;
   // UNI[4863] := 16#7EEF;
   // UNI[4864] := 16#7EF0;
   // UNI[4865] := 16#7EF1;
   // UNI[4866] := 16#7EF2;
   // UNI[4867] := 16#7EF3;
   // UNI[4868] := 16#7EF4;
   // UNI[4869] := 16#7EF5;
   // UNI[4870] := 16#7EF6;
   // UNI[4871] := 16#7EF7;
   // UNI[4872] := 16#7EF8;
   // UNI[4873] := 16#7EFA;
   // UNI[4874] := 16#7EFB;
   // UNI[4875] := 16#7EFC;
   // UNI[4876] := 16#7EFD;
   // UNI[4877] := 16#7EFE;
   // UNI[4878] := 16#7EFF;
   // UNI[4879] := 16#7F00;
   // UNI[4880] := 16#7F01;
   // UNI[4881] := 16#7F02;
   // UNI[4882] := 16#7F03;
   // UNI[4883] := 16#7F04;
   // UNI[4884] := 16#7F05;
   // UNI[4885] := 16#7F06;
   // UNI[4886] := 16#7F07;
   // UNI[4887] := 16#7F08;
   // UNI[4888] := 16#7F09;
   // UNI[4889] := 16#7F0B;
   // UNI[4890] := 16#7F0C;
   // UNI[4891] := 16#7F0D;
   // UNI[4892] := 16#7F0E;
   // UNI[4893] := 16#7F0F;
   // UNI[4894] := 16#7F11;
   // UNI[4895] := 16#7F12;
   // UNI[4896] := 16#7F13;
   // UNI[4897] := 16#7F14;
   // UNI[4898] := 16#7F15;
   // UNI[4899] := 16#7F16;
   // UNI[4900] := 16#7F17;
   // UNI[4901] := 16#7F18;
   // UNI[4902] := 16#7F19;
   // UNI[4903] := 16#7F1A;
   // UNI[4904] := 16#7F1B;
   // UNI[4905] := 16#7F1C;
   // UNI[4906] := 16#7F1D;
   // UNI[4907] := 16#7F1F;
   // UNI[4908] := 16#7F20;
   // UNI[4909] := 16#7F21;
   // UNI[4910] := 16#7F22;
   // UNI[4911] := 16#7F23;
   // UNI[4912] := 16#7F24;
   // UNI[4913] := 16#7F25;
   // UNI[4914] := 16#7F26;
   // UNI[4915] := 16#7F27;
   // UNI[4916] := 16#7F28;
   // UNI[4917] := 16#7F29;
   // UNI[4918] := 16#7F2A;
   // UNI[4919] := 16#7F2B;
   // UNI[4920] := 16#7F2C;
   // UNI[4921] := 16#7F2D;
   // UNI[4922] := 16#7F2E;
   // UNI[4923] := 16#7F2F;
   // UNI[4924] := 16#7F30;
   // UNI[4925] := 16#7F31;
   // UNI[4926] := 16#7F32;
   // UNI[4927] := 16#7F33;
   // UNI[4928] := 16#7F34;
   // UNI[4929] := 16#7F35;
   // UNI[4930] := 16#7F36;
   // UNI[4931] := 16#7F38;
   // UNI[4932] := 16#7F3A;
   // UNI[4933] := 16#7F42;
   // UNI[4934] := 16#7F44;
   // UNI[4935] := 16#7F45;
   // UNI[4936] := 16#7F50;
   // UNI[4937] := 16#7F51;
   // UNI[4938] := 16#7F54;
   // UNI[4939] := 16#7F55;
   // UNI[4940] := 16#7F57;
   // UNI[4941] := 16#7F58;
   // UNI[4942] := 16#7F5A;
   // UNI[4943] := 16#7F5F;
   // UNI[4944] := 16#7F61;
   // UNI[4945] := 16#7F62;
   // UNI[4946] := 16#7F68;
   // UNI[4947] := 16#7F69;
   // UNI[4948] := 16#7F6A;
   // UNI[4949] := 16#7F6E;
   // UNI[4950] := 16#7F71;
   // UNI[4951] := 16#7F72;
   // UNI[4952] := 16#7F74;
   // UNI[4953] := 16#7F79;
   // UNI[4954] := 16#7F7E;
   // UNI[4955] := 16#7F81;
   // UNI[4956] := 16#7F8A;
   // UNI[4957] := 16#7F8C;
   // UNI[4958] := 16#7F8E;
   // UNI[4959] := 16#7F94;
   // UNI[4960] := 16#7F9A;
   // UNI[4961] := 16#7F9D;
   // UNI[4962] := 16#7F9E;
   // UNI[4963] := 16#7F9F;
   // UNI[4964] := 16#7FA1;
   // UNI[4965] := 16#7FA4;
   // UNI[4966] := 16#7FA7;
   // UNI[4967] := 16#7FAF;
   // UNI[4968] := 16#7FB0;
   // UNI[4969] := 16#7FB2;
   // UNI[4970] := 16#7FB8;
   // UNI[4971] := 16#7FB9;
   // UNI[4972] := 16#7FBC;
   // UNI[4973] := 16#7FBD;
   // UNI[4974] := 16#7FBF;
   // UNI[4975] := 16#7FC1;
   // UNI[4976] := 16#7FC5;
   // UNI[4977] := 16#7FCA;
   // UNI[4978] := 16#7FCC;
   // UNI[4979] := 16#7FCE;
   // UNI[4980] := 16#7FD4;
   // UNI[4981] := 16#7FD5;
   // UNI[4982] := 16#7FD8;
   // UNI[4983] := 16#7FDF;
   // UNI[4984] := 16#7FE0;
   // UNI[4985] := 16#7FE1;
   // UNI[4986] := 16#7FE5;
   // UNI[4987] := 16#7FE6;
   // UNI[4988] := 16#7FE9;
   // UNI[4989] := 16#7FEE;
   // UNI[4990] := 16#7FF0;
   // UNI[4991] := 16#7FF1;
   // UNI[4992] := 16#7FF3;
   // UNI[4993] := 16#7FFB;
   // UNI[4994] := 16#7FFC;
   // UNI[4995] := 16#8000;
   // UNI[4996] := 16#8001;
   // UNI[4997] := 16#8003;
   // UNI[4998] := 16#8004;
   // UNI[4999] := 16#8005;
   // UNI[5000] := 16#8006;
   // UNI[5001] := 16#800B;
   // UNI[5002] := 16#800C;
   // UNI[5003] := 16#800D;
   // UNI[5004] := 16#8010;
   // UNI[5005] := 16#8012;
   // UNI[5006] := 16#8014;
   // UNI[5007] := 16#8015;
   // UNI[5008] := 16#8016;
   // UNI[5009] := 16#8017;
   // UNI[5010] := 16#8018;
   // UNI[5011] := 16#8019;
   // UNI[5012] := 16#801C;
   // UNI[5013] := 16#8020;
   // UNI[5014] := 16#8022;
   // UNI[5015] := 16#8025;
   // UNI[5016] := 16#8026;
   // UNI[5017] := 16#8027;
   // UNI[5018] := 16#8028;
   // UNI[5019] := 16#8029;
   // UNI[5020] := 16#802A;
   // UNI[5021] := 16#8031;
   // UNI[5022] := 16#8033;
   // UNI[5023] := 16#8035;
   // UNI[5024] := 16#8036;
   // UNI[5025] := 16#8037;
   // UNI[5026] := 16#8038;
   // UNI[5027] := 16#803B;
   // UNI[5028] := 16#803D;
   // UNI[5029] := 16#803F;
   // UNI[5030] := 16#8042;
   // UNI[5031] := 16#8043;
   // UNI[5032] := 16#8046;
   // UNI[5033] := 16#804A;
   // UNI[5034] := 16#804B;
   // UNI[5035] := 16#804C;
   // UNI[5036] := 16#804D;
   // UNI[5037] := 16#8052;
   // UNI[5038] := 16#8054;
   // UNI[5039] := 16#8058;
   // UNI[5040] := 16#805A;
   // UNI[5041] := 16#8069;
   // UNI[5042] := 16#806A;
   // UNI[5043] := 16#8071;
   // UNI[5044] := 16#807F;
   // UNI[5045] := 16#8080;
   // UNI[5046] := 16#8083;
   // UNI[5047] := 16#8084;
   // UNI[5048] := 16#8086;
   // UNI[5049] := 16#8087;
   // UNI[5050] := 16#8089;
   // UNI[5051] := 16#808B;
   // UNI[5052] := 16#808C;
   // UNI[5053] := 16#8093;
   // UNI[5054] := 16#8096;
   // UNI[5055] := 16#8098;
   // UNI[5056] := 16#809A;
   // UNI[5057] := 16#809B;
   // UNI[5058] := 16#809C;
   // UNI[5059] := 16#809D;
   // UNI[5060] := 16#809F;
   // UNI[5061] := 16#80A0;
   // UNI[5062] := 16#80A1;
   // UNI[5063] := 16#80A2;
   // UNI[5064] := 16#80A4;
   // UNI[5065] := 16#80A5;
   // UNI[5066] := 16#80A9;
   // UNI[5067] := 16#80AA;
   // UNI[5068] := 16#80AB;
   // UNI[5069] := 16#80AD;
   // UNI[5070] := 16#80AE;
   // UNI[5071] := 16#80AF;
   // UNI[5072] := 16#80B1;
   // UNI[5073] := 16#80B2;
   // UNI[5074] := 16#80B4;
   // UNI[5075] := 16#80B7;
   // UNI[5076] := 16#80BA;
   // UNI[5077] := 16#80BC;
   // UNI[5078] := 16#80BD;
   // UNI[5079] := 16#80BE;
   // UNI[5080] := 16#80BF;
   // UNI[5081] := 16#80C0;
   // UNI[5082] := 16#80C1;
   // UNI[5083] := 16#80C2;
   // UNI[5084] := 16#80C3;
   // UNI[5085] := 16#80C4;
   // UNI[5086] := 16#80C6;
   // UNI[5087] := 16#80CC;
   // UNI[5088] := 16#80CD;
   // UNI[5089] := 16#80CE;
   // UNI[5090] := 16#80D6;
   // UNI[5091] := 16#80D7;
   // UNI[5092] := 16#80D9;
   // UNI[5093] := 16#80DA;
   // UNI[5094] := 16#80DB;
   // UNI[5095] := 16#80DC;
   // UNI[5096] := 16#80DD;
   // UNI[5097] := 16#80DE;
   // UNI[5098] := 16#80E1;
   // UNI[5099] := 16#80E4;
   // UNI[5100] := 16#80E5;
   // UNI[5101] := 16#80E7;
   // UNI[5102] := 16#80E8;
   // UNI[5103] := 16#80E9;
   // UNI[5104] := 16#80EA;
   // UNI[5105] := 16#80EB;
   // UNI[5106] := 16#80EC;
   // UNI[5107] := 16#80ED;
   // UNI[5108] := 16#80EF;
   // UNI[5109] := 16#80F0;
   // UNI[5110] := 16#80F1;
   // UNI[5111] := 16#80F2;
   // UNI[5112] := 16#80F3;
   // UNI[5113] := 16#80F4;
   // UNI[5114] := 16#80F6;
   // UNI[5115] := 16#80F8;
   // UNI[5116] := 16#80FA;
   // UNI[5117] := 16#80FC;
   // UNI[5118] := 16#80FD;
   // UNI[5119] := 16#8102;
   // UNI[5120] := 16#8106;
   // UNI[5121] := 16#8109;
   // UNI[5122] := 16#810A;
   // UNI[5123] := 16#810D;
   // UNI[5124] := 16#810E;
   // UNI[5125] := 16#810F;
   // UNI[5126] := 16#8110;
   // UNI[5127] := 16#8111;
   // UNI[5128] := 16#8112;
   // UNI[5129] := 16#8113;
   // UNI[5130] := 16#8114;
   // UNI[5131] := 16#8116;
   // UNI[5132] := 16#8118;
   // UNI[5133] := 16#811A;
   // UNI[5134] := 16#811E;
   // UNI[5135] := 16#812C;
   // UNI[5136] := 16#812F;
   // UNI[5137] := 16#8131;
   // UNI[5138] := 16#8132;
   // UNI[5139] := 16#8136;
   // UNI[5140] := 16#8138;
   // UNI[5141] := 16#813E;
   // UNI[5142] := 16#8146;
   // UNI[5143] := 16#8148;
   // UNI[5144] := 16#814A;
   // UNI[5145] := 16#814B;
   // UNI[5146] := 16#814C;
   // UNI[5147] := 16#8150;
   // UNI[5148] := 16#8151;
   // UNI[5149] := 16#8153;
   // UNI[5150] := 16#8154;
   // UNI[5151] := 16#8155;
   // UNI[5152] := 16#8159;
   // UNI[5153] := 16#815A;
   // UNI[5154] := 16#8160;
   // UNI[5155] := 16#8165;
   // UNI[5156] := 16#8167;
   // UNI[5157] := 16#8169;
   // UNI[5158] := 16#816D;
   // UNI[5159] := 16#816E;
   // UNI[5160] := 16#8170;
   // UNI[5161] := 16#8171;
   // UNI[5162] := 16#8174;
   // UNI[5163] := 16#8179;
   // UNI[5164] := 16#817A;
   // UNI[5165] := 16#817B;
   // UNI[5166] := 16#817C;
   // UNI[5167] := 16#817D;
   // UNI[5168] := 16#817E;
   // UNI[5169] := 16#817F;
   // UNI[5170] := 16#8180;
   // UNI[5171] := 16#8182;
   // UNI[5172] := 16#8188;
   // UNI[5173] := 16#818A;
   // UNI[5174] := 16#818F;
   // UNI[5175] := 16#8191;
   // UNI[5176] := 16#8198;
   // UNI[5177] := 16#819B;
   // UNI[5178] := 16#819C;
   // UNI[5179] := 16#819D;
   // UNI[5180] := 16#81A3;
   // UNI[5181] := 16#81A6;
   // UNI[5182] := 16#81A8;
   // UNI[5183] := 16#81AA;
   // UNI[5184] := 16#81B3;
   // UNI[5185] := 16#81BA;
   // UNI[5186] := 16#81BB;
   // UNI[5187] := 16#81C0;
   // UNI[5188] := 16#81C1;
   // UNI[5189] := 16#81C2;
   // UNI[5190] := 16#81C3;
   // UNI[5191] := 16#81C6;
   // UNI[5192] := 16#81CA;
   // UNI[5193] := 16#81CC;
   // UNI[5194] := 16#81E3;
   // UNI[5195] := 16#81E7;
   // UNI[5196] := 16#81EA;
   // UNI[5197] := 16#81EC;
   // UNI[5198] := 16#81ED;
   // UNI[5199] := 16#81F3;
   // UNI[5200] := 16#81F4;
   // UNI[5201] := 16#81FB;
   // UNI[5202] := 16#81FC;
   // UNI[5203] := 16#81FE;
   // UNI[5204] := 16#8200;
   // UNI[5205] := 16#8201;
   // UNI[5206] := 16#8202;
   // UNI[5207] := 16#8204;
   // UNI[5208] := 16#8205;
   // UNI[5209] := 16#8206;
   // UNI[5210] := 16#820C;
   // UNI[5211] := 16#820D;
   // UNI[5212] := 16#8210;
   // UNI[5213] := 16#8212;
   // UNI[5214] := 16#8214;
   // UNI[5215] := 16#821B;
   // UNI[5216] := 16#821C;
   // UNI[5217] := 16#821E;
   // UNI[5218] := 16#821F;
   // UNI[5219] := 16#8221;
   // UNI[5220] := 16#8222;
   // UNI[5221] := 16#8223;
   // UNI[5222] := 16#8228;
   // UNI[5223] := 16#822A;
   // UNI[5224] := 16#822B;
   // UNI[5225] := 16#822C;
   // UNI[5226] := 16#822D;
   // UNI[5227] := 16#822F;
   // UNI[5228] := 16#8230;
   // UNI[5229] := 16#8231;
   // UNI[5230] := 16#8233;
   // UNI[5231] := 16#8234;
   // UNI[5232] := 16#8235;
   // UNI[5233] := 16#8236;
   // UNI[5234] := 16#8237;
   // UNI[5235] := 16#8238;
   // UNI[5236] := 16#8239;
   // UNI[5237] := 16#823B;
   // UNI[5238] := 16#823E;
   // UNI[5239] := 16#8244;
   // UNI[5240] := 16#8247;
   // UNI[5241] := 16#8249;
   // UNI[5242] := 16#824B;
   // UNI[5243] := 16#824F;
   // UNI[5244] := 16#8258;
   // UNI[5245] := 16#825A;
   // UNI[5246] := 16#825F;
   // UNI[5247] := 16#8268;
   // UNI[5248] := 16#826E;
   // UNI[5249] := 16#826F;
   // UNI[5250] := 16#8270;
   // UNI[5251] := 16#8272;
   // UNI[5252] := 16#8273;
   // UNI[5253] := 16#8274;
   // UNI[5254] := 16#8279;
   // UNI[5255] := 16#827A;
   // UNI[5256] := 16#827D;
   // UNI[5257] := 16#827E;
   // UNI[5258] := 16#827F;
   // UNI[5259] := 16#8282;
   // UNI[5260] := 16#8284;
   // UNI[5261] := 16#8288;
   // UNI[5262] := 16#828A;
   // UNI[5263] := 16#828B;
   // UNI[5264] := 16#828D;
   // UNI[5265] := 16#828E;
   // UNI[5266] := 16#828F;
   // UNI[5267] := 16#8291;
   // UNI[5268] := 16#8292;
   // UNI[5269] := 16#8297;
   // UNI[5270] := 16#8298;
   // UNI[5271] := 16#8299;
   // UNI[5272] := 16#829C;
   // UNI[5273] := 16#829D;
   // UNI[5274] := 16#829F;
   // UNI[5275] := 16#82A1;
   // UNI[5276] := 16#82A4;
   // UNI[5277] := 16#82A5;
   // UNI[5278] := 16#82A6;
   // UNI[5279] := 16#82A8;
   // UNI[5280] := 16#82A9;
   // UNI[5281] := 16#82AA;
   // UNI[5282] := 16#82AB;
   // UNI[5283] := 16#82AC;
   // UNI[5284] := 16#82AD;
   // UNI[5285] := 16#82AE;
   // UNI[5286] := 16#82AF;
   // UNI[5287] := 16#82B0;
   // UNI[5288] := 16#82B1;
   // UNI[5289] := 16#82B3;
   // UNI[5290] := 16#82B4;
   // UNI[5291] := 16#82B7;
   // UNI[5292] := 16#82B8;
   // UNI[5293] := 16#82B9;
   // UNI[5294] := 16#82BD;
   // UNI[5295] := 16#82BE;
   // UNI[5296] := 16#82C1;
   // UNI[5297] := 16#82C4;
   // UNI[5298] := 16#82C7;
   // UNI[5299] := 16#82C8;
   // UNI[5300] := 16#82CA;
   // UNI[5301] := 16#82CB;
   // UNI[5302] := 16#82CC;
   // UNI[5303] := 16#82CD;
   // UNI[5304] := 16#82CE;
   // UNI[5305] := 16#82CF;
   // UNI[5306] := 16#82D1;
   // UNI[5307] := 16#82D2;
   // UNI[5308] := 16#82D3;
   // UNI[5309] := 16#82D4;
   // UNI[5310] := 16#82D5;
   // UNI[5311] := 16#82D7;
   // UNI[5312] := 16#82D8;
   // UNI[5313] := 16#82DB;
   // UNI[5314] := 16#82DC;
   // UNI[5315] := 16#82DE;
   // UNI[5316] := 16#82DF;
   // UNI[5317] := 16#82E0;
   // UNI[5318] := 16#82E1;
   // UNI[5319] := 16#82E3;
   // UNI[5320] := 16#82E4;
   // UNI[5321] := 16#82E5;
   // UNI[5322] := 16#82E6;
   // UNI[5323] := 16#82EB;
   // UNI[5324] := 16#82EF;
   // UNI[5325] := 16#82F1;
   // UNI[5326] := 16#82F4;
   // UNI[5327] := 16#82F7;
   // UNI[5328] := 16#82F9;
   // UNI[5329] := 16#82FB;
   // UNI[5330] := 16#8301;
   // UNI[5331] := 16#8302;
   // UNI[5332] := 16#8303;
   // UNI[5333] := 16#8304;
   // UNI[5334] := 16#8305;
   // UNI[5335] := 16#8306;
   // UNI[5336] := 16#8307;
   // UNI[5337] := 16#8308;
   // UNI[5338] := 16#8309;
   // UNI[5339] := 16#830C;
   // UNI[5340] := 16#830E;
   // UNI[5341] := 16#830F;
   // UNI[5342] := 16#8311;
   // UNI[5343] := 16#8314;
   // UNI[5344] := 16#8315;
   // UNI[5345] := 16#8317;
   // UNI[5346] := 16#831A;
   // UNI[5347] := 16#831B;
   // UNI[5348] := 16#831C;
   // UNI[5349] := 16#8327;
   // UNI[5350] := 16#8328;
   // UNI[5351] := 16#832B;
   // UNI[5352] := 16#832C;
   // UNI[5353] := 16#832D;
   // UNI[5354] := 16#832F;
   // UNI[5355] := 16#8331;
   // UNI[5356] := 16#8333;
   // UNI[5357] := 16#8334;
   // UNI[5358] := 16#8335;
   // UNI[5359] := 16#8336;
   // UNI[5360] := 16#8338;
   // UNI[5361] := 16#8339;
   // UNI[5362] := 16#833A;
   // UNI[5363] := 16#833C;
   // UNI[5364] := 16#8340;
   // UNI[5365] := 16#8343;
   // UNI[5366] := 16#8346;
   // UNI[5367] := 16#8347;
   // UNI[5368] := 16#8349;
   // UNI[5369] := 16#834F;
   // UNI[5370] := 16#8350;
   // UNI[5371] := 16#8351;
   // UNI[5372] := 16#8352;
   // UNI[5373] := 16#8354;
   // UNI[5374] := 16#835A;
   // UNI[5375] := 16#835B;
   // UNI[5376] := 16#835C;
   // UNI[5377] := 16#835E;
   // UNI[5378] := 16#835F;
   // UNI[5379] := 16#8360;
   // UNI[5380] := 16#8361;
   // UNI[5381] := 16#8363;
   // UNI[5382] := 16#8364;
   // UNI[5383] := 16#8365;
   // UNI[5384] := 16#8366;
   // UNI[5385] := 16#8367;
   // UNI[5386] := 16#8368;
   // UNI[5387] := 16#8369;
   // UNI[5388] := 16#836A;
   // UNI[5389] := 16#836B;
   // UNI[5390] := 16#836C;
   // UNI[5391] := 16#836D;
   // UNI[5392] := 16#836E;
   // UNI[5393] := 16#836F;
   // UNI[5394] := 16#8377;
   // UNI[5395] := 16#8378;
   // UNI[5396] := 16#837B;
   // UNI[5397] := 16#837C;
   // UNI[5398] := 16#837D;
   // UNI[5399] := 16#8385;
   // UNI[5400] := 16#8386;
   // UNI[5401] := 16#8389;
   // UNI[5402] := 16#838E;
   // UNI[5403] := 16#8392;
   // UNI[5404] := 16#8393;
   // UNI[5405] := 16#8398;
   // UNI[5406] := 16#839B;
   // UNI[5407] := 16#839C;
   // UNI[5408] := 16#839E;
   // UNI[5409] := 16#83A0;
   // UNI[5410] := 16#83A8;
   // UNI[5411] := 16#83A9;
   // UNI[5412] := 16#83AA;
   // UNI[5413] := 16#83AB;
   // UNI[5414] := 16#83B0;
   // UNI[5415] := 16#83B1;
   // UNI[5416] := 16#83B2;
   // UNI[5417] := 16#83B3;
   // UNI[5418] := 16#83B4;
   // UNI[5419] := 16#83B6;
   // UNI[5420] := 16#83B7;
   // UNI[5421] := 16#83B8;
   // UNI[5422] := 16#83B9;
   // UNI[5423] := 16#83BA;
   // UNI[5424] := 16#83BC;
   // UNI[5425] := 16#83BD;
   // UNI[5426] := 16#83C0;
   // UNI[5427] := 16#83C1;
   // UNI[5428] := 16#83C5;
   // UNI[5429] := 16#83C7;
   // UNI[5430] := 16#83CA;
   // UNI[5431] := 16#83CC;
   // UNI[5432] := 16#83CF;
   // UNI[5433] := 16#83D4;
   // UNI[5434] := 16#83D6;
   // UNI[5435] := 16#83D8;
   // UNI[5436] := 16#83DC;
   // UNI[5437] := 16#83DD;
   // UNI[5438] := 16#83DF;
   // UNI[5439] := 16#83E0;
   // UNI[5440] := 16#83E1;
   // UNI[5441] := 16#83E5;
   // UNI[5442] := 16#83E9;
   // UNI[5443] := 16#83EA;
   // UNI[5444] := 16#83F0;
   // UNI[5445] := 16#83F1;
   // UNI[5446] := 16#83F2;
   // UNI[5447] := 16#83F8;
   // UNI[5448] := 16#83F9;
   // UNI[5449] := 16#83FD;
   // UNI[5450] := 16#8401;
   // UNI[5451] := 16#8403;
   // UNI[5452] := 16#8404;
   // UNI[5453] := 16#8406;
   // UNI[5454] := 16#840B;
   // UNI[5455] := 16#840C;
   // UNI[5456] := 16#840D;
   // UNI[5457] := 16#840E;
   // UNI[5458] := 16#840F;
   // UNI[5459] := 16#8411;
   // UNI[5460] := 16#8418;
   // UNI[5461] := 16#841C;
   // UNI[5462] := 16#841D;
   // UNI[5463] := 16#8424;
   // UNI[5464] := 16#8425;
   // UNI[5465] := 16#8426;
   // UNI[5466] := 16#8427;
   // UNI[5467] := 16#8428;
   // UNI[5468] := 16#8431;
   // UNI[5469] := 16#8438;
   // UNI[5470] := 16#843C;
   // UNI[5471] := 16#843D;
   // UNI[5472] := 16#8446;
   // UNI[5473] := 16#8451;
   // UNI[5474] := 16#8457;
   // UNI[5475] := 16#8459;
   // UNI[5476] := 16#845A;
   // UNI[5477] := 16#845B;
   // UNI[5478] := 16#845C;
   // UNI[5479] := 16#8461;
   // UNI[5480] := 16#8463;
   // UNI[5481] := 16#8469;
   // UNI[5482] := 16#846B;
   // UNI[5483] := 16#846C;
   // UNI[5484] := 16#846D;
   // UNI[5485] := 16#8471;
   // UNI[5486] := 16#8473;
   // UNI[5487] := 16#8475;
   // UNI[5488] := 16#8476;
   // UNI[5489] := 16#8478;
   // UNI[5490] := 16#847A;
   // UNI[5491] := 16#8482;
   // UNI[5492] := 16#8487;
   // UNI[5493] := 16#8488;
   // UNI[5494] := 16#8489;
   // UNI[5495] := 16#848B;
   // UNI[5496] := 16#848C;
   // UNI[5497] := 16#848E;
   // UNI[5498] := 16#8497;
   // UNI[5499] := 16#8499;
   // UNI[5500] := 16#849C;
   // UNI[5501] := 16#84A1;
   // UNI[5502] := 16#84AF;
   // UNI[5503] := 16#84B2;
   // UNI[5504] := 16#84B4;
   // UNI[5505] := 16#84B8;
   // UNI[5506] := 16#84B9;
   // UNI[5507] := 16#84BA;
   // UNI[5508] := 16#84BD;
   // UNI[5509] := 16#84BF;
   // UNI[5510] := 16#84C1;
   // UNI[5511] := 16#84C4;
   // UNI[5512] := 16#84C9;
   // UNI[5513] := 16#84CA;
   // UNI[5514] := 16#84CD;
   // UNI[5515] := 16#84D0;
   // UNI[5516] := 16#84D1;
   // UNI[5517] := 16#84D3;
   // UNI[5518] := 16#84D6;
   // UNI[5519] := 16#84DD;
   // UNI[5520] := 16#84DF;
   // UNI[5521] := 16#84E0;
   // UNI[5522] := 16#84E3;
   // UNI[5523] := 16#84E5;
   // UNI[5524] := 16#84E6;
   // UNI[5525] := 16#84EC;
   // UNI[5526] := 16#84F0;
   // UNI[5527] := 16#84FC;
   // UNI[5528] := 16#84FF;
   // UNI[5529] := 16#850C;
   // UNI[5530] := 16#8511;
   // UNI[5531] := 16#8513;
   // UNI[5532] := 16#8517;
   // UNI[5533] := 16#851A;
   // UNI[5534] := 16#851F;
   // UNI[5535] := 16#8521;
   // UNI[5536] := 16#852B;
   // UNI[5537] := 16#852C;
   // UNI[5538] := 16#8537;
   // UNI[5539] := 16#8538;
   // UNI[5540] := 16#8539;
   // UNI[5541] := 16#853A;
   // UNI[5542] := 16#853B;
   // UNI[5543] := 16#853C;
   // UNI[5544] := 16#853D;
   // UNI[5545] := 16#8543;
   // UNI[5546] := 16#8548;
   // UNI[5547] := 16#8549;
   // UNI[5548] := 16#854A;
   // UNI[5549] := 16#8556;
   // UNI[5550] := 16#8559;
   // UNI[5551] := 16#855E;
   // UNI[5552] := 16#8564;
   // UNI[5553] := 16#8568;
   // UNI[5554] := 16#8572;
   // UNI[5555] := 16#8574;
   // UNI[5556] := 16#8579;
   // UNI[5557] := 16#857A;
   // UNI[5558] := 16#857B;
   // UNI[5559] := 16#857E;
   // UNI[5560] := 16#8584;
   // UNI[5561] := 16#8585;
   // UNI[5562] := 16#8587;
   // UNI[5563] := 16#858F;
   // UNI[5564] := 16#859B;
   // UNI[5565] := 16#859C;
   // UNI[5566] := 16#85A4;
   // UNI[5567] := 16#85A8;
   // UNI[5568] := 16#85AA;
   // UNI[5569] := 16#85AE;
   // UNI[5570] := 16#85AF;
   // UNI[5571] := 16#85B0;
   // UNI[5572] := 16#85B7;
   // UNI[5573] := 16#85B9;
   // UNI[5574] := 16#85C1;
   // UNI[5575] := 16#85C9;
   // UNI[5576] := 16#85CF;
   // UNI[5577] := 16#85D0;
   // UNI[5578] := 16#85D3;
   // UNI[5579] := 16#85D5;
   // UNI[5580] := 16#85DC;
   // UNI[5581] := 16#85E4;
   // UNI[5582] := 16#85E9;
   // UNI[5583] := 16#85FB;
   // UNI[5584] := 16#85FF;
   // UNI[5585] := 16#8605;
   // UNI[5586] := 16#8611;
   // UNI[5587] := 16#8616;
   // UNI[5588] := 16#8627;
   // UNI[5589] := 16#8629;
   // UNI[5590] := 16#8638;
   // UNI[5591] := 16#863C;
   // UNI[5592] := 16#864D;
   // UNI[5593] := 16#864E;
   // UNI[5594] := 16#864F;
   // UNI[5595] := 16#8650;
   // UNI[5596] := 16#8651;
   // UNI[5597] := 16#8654;
   // UNI[5598] := 16#865A;
   // UNI[5599] := 16#865E;
   // UNI[5600] := 16#8662;
   // UNI[5601] := 16#866B;
   // UNI[5602] := 16#866C;
   // UNI[5603] := 16#866E;
   // UNI[5604] := 16#8671;
   // UNI[5605] := 16#8679;
   // UNI[5606] := 16#867A;
   // UNI[5607] := 16#867B;
   // UNI[5608] := 16#867C;
   // UNI[5609] := 16#867D;
   // UNI[5610] := 16#867E;
   // UNI[5611] := 16#867F;
   // UNI[5612] := 16#8680;
   // UNI[5613] := 16#8681;
   // UNI[5614] := 16#8682;
   // UNI[5615] := 16#868A;
   // UNI[5616] := 16#868B;
   // UNI[5617] := 16#868C;
   // UNI[5618] := 16#868D;
   // UNI[5619] := 16#8693;
   // UNI[5620] := 16#8695;
   // UNI[5621] := 16#869C;
   // UNI[5622] := 16#869D;
   // UNI[5623] := 16#86A3;
   // UNI[5624] := 16#86A4;
   // UNI[5625] := 16#86A7;
   // UNI[5626] := 16#86A8;
   // UNI[5627] := 16#86A9;
   // UNI[5628] := 16#86AA;
   // UNI[5629] := 16#86AC;
   // UNI[5630] := 16#86AF;
   // UNI[5631] := 16#86B0;
   // UNI[5632] := 16#86B1;
   // UNI[5633] := 16#86B4;
   // UNI[5634] := 16#86B5;
   // UNI[5635] := 16#86B6;
   // UNI[5636] := 16#86BA;
   // UNI[5637] := 16#86C0;
   // UNI[5638] := 16#86C4;
   // UNI[5639] := 16#86C6;
   // UNI[5640] := 16#86C7;
   // UNI[5641] := 16#86C9;
   // UNI[5642] := 16#86CA;
   // UNI[5643] := 16#86CB;
   // UNI[5644] := 16#86CE;
   // UNI[5645] := 16#86CF;
   // UNI[5646] := 16#86D0;
   // UNI[5647] := 16#86D1;
   // UNI[5648] := 16#86D4;
   // UNI[5649] := 16#86D8;
   // UNI[5650] := 16#86D9;
   // UNI[5651] := 16#86DB;
   // UNI[5652] := 16#86DE;
   // UNI[5653] := 16#86DF;
   // UNI[5654] := 16#86E4;
   // UNI[5655] := 16#86E9;
   // UNI[5656] := 16#86ED;
   // UNI[5657] := 16#86EE;
   // UNI[5658] := 16#86F0;
   // UNI[5659] := 16#86F1;
   // UNI[5660] := 16#86F2;
   // UNI[5661] := 16#86F3;
   // UNI[5662] := 16#86F4;
   // UNI[5663] := 16#86F8;
   // UNI[5664] := 16#86F9;
   // UNI[5665] := 16#86FE;
   // UNI[5666] := 16#8700;
   // UNI[5667] := 16#8702;
   // UNI[5668] := 16#8703;
   // UNI[5669] := 16#8707;
   // UNI[5670] := 16#8708;
   // UNI[5671] := 16#8709;
   // UNI[5672] := 16#870A;
   // UNI[5673] := 16#870D;
   // UNI[5674] := 16#8712;
   // UNI[5675] := 16#8713;
   // UNI[5676] := 16#8715;
   // UNI[5677] := 16#8717;
   // UNI[5678] := 16#8718;
   // UNI[5679] := 16#871A;
   // UNI[5680] := 16#871C;
   // UNI[5681] := 16#871E;
   // UNI[5682] := 16#8721;
   // UNI[5683] := 16#8722;
   // UNI[5684] := 16#8723;
   // UNI[5685] := 16#8725;
   // UNI[5686] := 16#8729;
   // UNI[5687] := 16#872E;
   // UNI[5688] := 16#8731;
   // UNI[5689] := 16#8734;
   // UNI[5690] := 16#8737;
   // UNI[5691] := 16#873B;
   // UNI[5692] := 16#873E;
   // UNI[5693] := 16#873F;
   // UNI[5694] := 16#8747;
   // UNI[5695] := 16#8748;
   // UNI[5696] := 16#8749;
   // UNI[5697] := 16#874C;
   // UNI[5698] := 16#874E;
   // UNI[5699] := 16#8753;
   // UNI[5700] := 16#8757;
   // UNI[5701] := 16#8759;
   // UNI[5702] := 16#8760;
   // UNI[5703] := 16#8763;
   // UNI[5704] := 16#8764;
   // UNI[5705] := 16#8765;
   // UNI[5706] := 16#876E;
   // UNI[5707] := 16#8770;
   // UNI[5708] := 16#8774;
   // UNI[5709] := 16#8776;
   // UNI[5710] := 16#877B;
   // UNI[5711] := 16#877C;
   // UNI[5712] := 16#877D;
   // UNI[5713] := 16#877E;
   // UNI[5714] := 16#8782;
   // UNI[5715] := 16#8783;
   // UNI[5716] := 16#8785;
   // UNI[5717] := 16#8788;
   // UNI[5718] := 16#878B;
   // UNI[5719] := 16#878D;
   // UNI[5720] := 16#8793;
   // UNI[5721] := 16#8797;
   // UNI[5722] := 16#879F;
   // UNI[5723] := 16#87A8;
   // UNI[5724] := 16#87AB;
   // UNI[5725] := 16#87AC;
   // UNI[5726] := 16#87AD;
   // UNI[5727] := 16#87AF;
   // UNI[5728] := 16#87B3;
   // UNI[5729] := 16#87B5;
   // UNI[5730] := 16#87BA;
   // UNI[5731] := 16#87BD;
   // UNI[5732] := 16#87C0;
   // UNI[5733] := 16#87C6;
   // UNI[5734] := 16#87CA;
   // UNI[5735] := 16#87CB;
   // UNI[5736] := 16#87D1;
   // UNI[5737] := 16#87D2;
   // UNI[5738] := 16#87D3;
   // UNI[5739] := 16#87DB;
   // UNI[5740] := 16#87E0;
   // UNI[5741] := 16#87E5;
   // UNI[5742] := 16#87EA;
   // UNI[5743] := 16#87EE;
   // UNI[5744] := 16#87F9;
   // UNI[5745] := 16#87FE;
   // UNI[5746] := 16#8803;
   // UNI[5747] := 16#880A;
   // UNI[5748] := 16#8813;
   // UNI[5749] := 16#8815;
   // UNI[5750] := 16#8816;
   // UNI[5751] := 16#881B;
   // UNI[5752] := 16#8821;
   // UNI[5753] := 16#8822;
   // UNI[5754] := 16#8832;
   // UNI[5755] := 16#8839;
   // UNI[5756] := 16#883C;
   // UNI[5757] := 16#8840;
   // UNI[5758] := 16#8844;
   // UNI[5759] := 16#8845;
   // UNI[5760] := 16#884C;
   // UNI[5761] := 16#884D;
   // UNI[5762] := 16#8854;
   // UNI[5763] := 16#8857;
   // UNI[5764] := 16#8859;
   // UNI[5765] := 16#8861;
   // UNI[5766] := 16#8862;
   // UNI[5767] := 16#8863;
   // UNI[5768] := 16#8864;
   // UNI[5769] := 16#8865;
   // UNI[5770] := 16#8868;
   // UNI[5771] := 16#8869;
   // UNI[5772] := 16#886B;
   // UNI[5773] := 16#886C;
   // UNI[5774] := 16#886E;
   // UNI[5775] := 16#8870;
   // UNI[5776] := 16#8872;
   // UNI[5777] := 16#8877;
   // UNI[5778] := 16#887D;
   // UNI[5779] := 16#887E;
   // UNI[5780] := 16#887F;
   // UNI[5781] := 16#8881;
   // UNI[5782] := 16#8882;
   // UNI[5783] := 16#8884;
   // UNI[5784] := 16#8885;
   // UNI[5785] := 16#8888;
   // UNI[5786] := 16#888B;
   // UNI[5787] := 16#888D;
   // UNI[5788] := 16#8892;
   // UNI[5789] := 16#8896;
   // UNI[5790] := 16#889C;
   // UNI[5791] := 16#88A2;
   // UNI[5792] := 16#88A4;
   // UNI[5793] := 16#88AB;
   // UNI[5794] := 16#88AD;
   // UNI[5795] := 16#88B1;
   // UNI[5796] := 16#88B7;
   // UNI[5797] := 16#88BC;
   // UNI[5798] := 16#88C1;
   // UNI[5799] := 16#88C2;
   // UNI[5800] := 16#88C5;
   // UNI[5801] := 16#88C6;
   // UNI[5802] := 16#88C9;
   // UNI[5803] := 16#88CE;
   // UNI[5804] := 16#88D2;
   // UNI[5805] := 16#88D4;
   // UNI[5806] := 16#88D5;
   // UNI[5807] := 16#88D8;
   // UNI[5808] := 16#88D9;
   // UNI[5809] := 16#88DF;
   // UNI[5810] := 16#88E2;
   // UNI[5811] := 16#88E3;
   // UNI[5812] := 16#88E4;
   // UNI[5813] := 16#88E5;
   // UNI[5814] := 16#88E8;
   // UNI[5815] := 16#88F0;
   // UNI[5816] := 16#88F1;
   // UNI[5817] := 16#88F3;
   // UNI[5818] := 16#88F4;
   // UNI[5819] := 16#88F8;
   // UNI[5820] := 16#88F9;
   // UNI[5821] := 16#88FC;
   // UNI[5822] := 16#88FE;
   // UNI[5823] := 16#8902;
   // UNI[5824] := 16#890A;
   // UNI[5825] := 16#8910;
   // UNI[5826] := 16#8912;
   // UNI[5827] := 16#8913;
   // UNI[5828] := 16#8919;
   // UNI[5829] := 16#891A;
   // UNI[5830] := 16#891B;
   // UNI[5831] := 16#8921;
   // UNI[5832] := 16#8925;
   // UNI[5833] := 16#892A;
   // UNI[5834] := 16#892B;
   // UNI[5835] := 16#8930;
   // UNI[5836] := 16#8934;
   // UNI[5837] := 16#8936;
   // UNI[5838] := 16#8941;
   // UNI[5839] := 16#8944;
   // UNI[5840] := 16#895E;
   // UNI[5841] := 16#895F;
   // UNI[5842] := 16#8966;
   // UNI[5843] := 16#897B;
   // UNI[5844] := 16#897F;
   // UNI[5845] := 16#8981;
   // UNI[5846] := 16#8983;
   // UNI[5847] := 16#8986;
   // UNI[5848] := 16#89C1;
   // UNI[5849] := 16#89C2;
   // UNI[5850] := 16#89C4;
   // UNI[5851] := 16#89C5;
   // UNI[5852] := 16#89C6;
   // UNI[5853] := 16#89C7;
   // UNI[5854] := 16#89C8;
   // UNI[5855] := 16#89C9;
   // UNI[5856] := 16#89CA;
   // UNI[5857] := 16#89CB;
   // UNI[5858] := 16#89CC;
   // UNI[5859] := 16#89CE;
   // UNI[5860] := 16#89CF;
   // UNI[5861] := 16#89D0;
   // UNI[5862] := 16#89D1;
   // UNI[5863] := 16#89D2;
   // UNI[5864] := 16#89D6;
   // UNI[5865] := 16#89DA;
   // UNI[5866] := 16#89DC;
   // UNI[5867] := 16#89DE;
   // UNI[5868] := 16#89E3;
   // UNI[5869] := 16#89E5;
   // UNI[5870] := 16#89E6;
   // UNI[5871] := 16#89EB;
   // UNI[5872] := 16#89EF;
   // UNI[5873] := 16#89F3;
   // UNI[5874] := 16#8A00;
   // UNI[5875] := 16#8A07;
   // UNI[5876] := 16#8A3E;
   // UNI[5877] := 16#8A48;
   // UNI[5878] := 16#8A79;
   // UNI[5879] := 16#8A89;
   // UNI[5880] := 16#8A8A;
   // UNI[5881] := 16#8A93;
   // UNI[5882] := 16#8B07;
   // UNI[5883] := 16#8B26;
   // UNI[5884] := 16#8B66;
   // UNI[5885] := 16#8B6C;
   // UNI[5886] := 16#8BA0;
   // UNI[5887] := 16#8BA1;
   // UNI[5888] := 16#8BA2;
   // UNI[5889] := 16#8BA3;
   // UNI[5890] := 16#8BA4;
   // UNI[5891] := 16#8BA5;
   // UNI[5892] := 16#8BA6;
   // UNI[5893] := 16#8BA7;
   // UNI[5894] := 16#8BA8;
   // UNI[5895] := 16#8BA9;
   // UNI[5896] := 16#8BAA;
   // UNI[5897] := 16#8BAB;
   // UNI[5898] := 16#8BAD;
   // UNI[5899] := 16#8BAE;
   // UNI[5900] := 16#8BAF;
   // UNI[5901] := 16#8BB0;
   // UNI[5902] := 16#8BB2;
   // UNI[5903] := 16#8BB3;
   // UNI[5904] := 16#8BB4;
   // UNI[5905] := 16#8BB5;
   // UNI[5906] := 16#8BB6;
   // UNI[5907] := 16#8BB7;
   // UNI[5908] := 16#8BB8;
   // UNI[5909] := 16#8BB9;
   // UNI[5910] := 16#8BBA;
   // UNI[5911] := 16#8BBC;
   // UNI[5912] := 16#8BBD;
   // UNI[5913] := 16#8BBE;
   // UNI[5914] := 16#8BBF;
   // UNI[5915] := 16#8BC0;
   // UNI[5916] := 16#8BC1;
   // UNI[5917] := 16#8BC2;
   // UNI[5918] := 16#8BC3;
   // UNI[5919] := 16#8BC4;
   // UNI[5920] := 16#8BC5;
   // UNI[5921] := 16#8BC6;
   // UNI[5922] := 16#8BC8;
   // UNI[5923] := 16#8BC9;
   // UNI[5924] := 16#8BCA;
   // UNI[5925] := 16#8BCB;
   // UNI[5926] := 16#8BCC;
   // UNI[5927] := 16#8BCD;
   // UNI[5928] := 16#8BCE;
   // UNI[5929] := 16#8BCF;
   // UNI[5930] := 16#8BD1;
   // UNI[5931] := 16#8BD2;
   // UNI[5932] := 16#8BD3;
   // UNI[5933] := 16#8BD4;
   // UNI[5934] := 16#8BD5;
   // UNI[5935] := 16#8BD6;
   // UNI[5936] := 16#8BD7;
   // UNI[5937] := 16#8BD8;
   // UNI[5938] := 16#8BD9;
   // UNI[5939] := 16#8BDA;
   // UNI[5940] := 16#8BDB;
   // UNI[5941] := 16#8BDC;
   // UNI[5942] := 16#8BDD;
   // UNI[5943] := 16#8BDE;
   // UNI[5944] := 16#8BDF;
   // UNI[5945] := 16#8BE0;
   // UNI[5946] := 16#8BE1;
   // UNI[5947] := 16#8BE2;
   // UNI[5948] := 16#8BE3;
   // UNI[5949] := 16#8BE4;
   // UNI[5950] := 16#8BE5;
   // UNI[5951] := 16#8BE6;
   // UNI[5952] := 16#8BE7;
   // UNI[5953] := 16#8BE8;
   // UNI[5954] := 16#8BE9;
   // UNI[5955] := 16#8BEB;
   // UNI[5956] := 16#8BEC;
   // UNI[5957] := 16#8BED;
   // UNI[5958] := 16#8BEE;
   // UNI[5959] := 16#8BEF;
   // UNI[5960] := 16#8BF0;
   // UNI[5961] := 16#8BF1;
   // UNI[5962] := 16#8BF2;
   // UNI[5963] := 16#8BF3;
   // UNI[5964] := 16#8BF4;
   // UNI[5965] := 16#8BF5;
   // UNI[5966] := 16#8BF6;
   // UNI[5967] := 16#8BF7;
   // UNI[5968] := 16#8BF8;
   // UNI[5969] := 16#8BF9;
   // UNI[5970] := 16#8BFA;
   // UNI[5971] := 16#8BFB;
   // UNI[5972] := 16#8BFC;
   // UNI[5973] := 16#8BFD;
   // UNI[5974] := 16#8BFE;
   // UNI[5975] := 16#8BFF;
   // UNI[5976] := 16#8C00;
   // UNI[5977] := 16#8C01;
   // UNI[5978] := 16#8C02;
   // UNI[5979] := 16#8C03;
   // UNI[5980] := 16#8C04;
   // UNI[5981] := 16#8C05;
   // UNI[5982] := 16#8C06;
   // UNI[5983] := 16#8C07;
   // UNI[5984] := 16#8C08;
   // UNI[5985] := 16#8C0A;
   // UNI[5986] := 16#8C0B;
   // UNI[5987] := 16#8C0C;
   // UNI[5988] := 16#8C0D;
   // UNI[5989] := 16#8C0E;
   // UNI[5990] := 16#8C0F;
   // UNI[5991] := 16#8C10;
   // UNI[5992] := 16#8C11;
   // UNI[5993] := 16#8C12;
   // UNI[5994] := 16#8C13;
   // UNI[5995] := 16#8C14;
   // UNI[5996] := 16#8C15;
   // UNI[5997] := 16#8C16;
   // UNI[5998] := 16#8C17;
   // UNI[5999] := 16#8C18;
   // UNI[6000] := 16#8C19;
   // UNI[6001] := 16#8C1A;
   // UNI[6002] := 16#8C1B;
   // UNI[6003] := 16#8C1C;
   // UNI[6004] := 16#8C1D;
   // UNI[6005] := 16#8C1F;
   // UNI[6006] := 16#8C20;
   // UNI[6007] := 16#8C21;
   // UNI[6008] := 16#8C22;
   // UNI[6009] := 16#8C23;
   // UNI[6010] := 16#8C24;
   // UNI[6011] := 16#8C25;
   // UNI[6012] := 16#8C26;
   // UNI[6013] := 16#8C27;
   // UNI[6014] := 16#8C28;
   // UNI[6015] := 16#8C29;
   // UNI[6016] := 16#8C2A;
   // UNI[6017] := 16#8C2B;
   // UNI[6018] := 16#8C2C;
   // UNI[6019] := 16#8C2D;
   // UNI[6020] := 16#8C2E;
   // UNI[6021] := 16#8C2F;
   // UNI[6022] := 16#8C30;
   // UNI[6023] := 16#8C31;
   // UNI[6024] := 16#8C32;
   // UNI[6025] := 16#8C33;
   // UNI[6026] := 16#8C34;
   // UNI[6027] := 16#8C35;
   // UNI[6028] := 16#8C36;
   // UNI[6029] := 16#8C37;
   // UNI[6030] := 16#8C41;
   // UNI[6031] := 16#8C46;
   // UNI[6032] := 16#8C47;
   // UNI[6033] := 16#8C49;
   // UNI[6034] := 16#8C4C;
   // UNI[6035] := 16#8C55;
   // UNI[6036] := 16#8C5A;
   // UNI[6037] := 16#8C61;
   // UNI[6038] := 16#8C62;
   // UNI[6039] := 16#8C6A;
   // UNI[6040] := 16#8C6B;
   // UNI[6041] := 16#8C73;
   // UNI[6042] := 16#8C78;
   // UNI[6043] := 16#8C79;
   // UNI[6044] := 16#8C7A;
   // UNI[6045] := 16#8C82;
   // UNI[6046] := 16#8C85;
   // UNI[6047] := 16#8C89;
   // UNI[6048] := 16#8C8A;
   // UNI[6049] := 16#8C8C;
   // UNI[6050] := 16#8C94;
   // UNI[6051] := 16#8C98;
   // UNI[6052] := 16#8D1D;
   // UNI[6053] := 16#8D1E;
   // UNI[6054] := 16#8D1F;
   // UNI[6055] := 16#8D21;
   // UNI[6056] := 16#8D22;
   // UNI[6057] := 16#8D23;
   // UNI[6058] := 16#8D24;
   // UNI[6059] := 16#8D25;
   // UNI[6060] := 16#8D26;
   // UNI[6061] := 16#8D27;
   // UNI[6062] := 16#8D28;
   // UNI[6063] := 16#8D29;
   // UNI[6064] := 16#8D2A;
   // UNI[6065] := 16#8D2B;
   // UNI[6066] := 16#8D2C;
   // UNI[6067] := 16#8D2D;
   // UNI[6068] := 16#8D2E;
   // UNI[6069] := 16#8D2F;
   // UNI[6070] := 16#8D30;
   // UNI[6071] := 16#8D31;
   // UNI[6072] := 16#8D32;
   // UNI[6073] := 16#8D33;
   // UNI[6074] := 16#8D34;
   // UNI[6075] := 16#8D35;
   // UNI[6076] := 16#8D36;
   // UNI[6077] := 16#8D37;
   // UNI[6078] := 16#8D38;
   // UNI[6079] := 16#8D39;
   // UNI[6080] := 16#8D3A;
   // UNI[6081] := 16#8D3B;
   // UNI[6082] := 16#8D3C;
   // UNI[6083] := 16#8D3D;
   // UNI[6084] := 16#8D3E;
   // UNI[6085] := 16#8D3F;
   // UNI[6086] := 16#8D40;
   // UNI[6087] := 16#8D41;
   // UNI[6088] := 16#8D42;
   // UNI[6089] := 16#8D43;
   // UNI[6090] := 16#8D44;
   // UNI[6091] := 16#8D45;
   // UNI[6092] := 16#8D46;
   // UNI[6093] := 16#8D47;
   // UNI[6094] := 16#8D48;
   // UNI[6095] := 16#8D49;
   // UNI[6096] := 16#8D4A;
   // UNI[6097] := 16#8D4B;
   // UNI[6098] := 16#8D4C;
   // UNI[6099] := 16#8D4D;
   // UNI[6100] := 16#8D4E;
   // UNI[6101] := 16#8D4F;
   // UNI[6102] := 16#8D50;
   // UNI[6103] := 16#8D53;
   // UNI[6104] := 16#8D54;
   // UNI[6105] := 16#8D55;
   // UNI[6106] := 16#8D56;
   // UNI[6107] := 16#8D58;
   // UNI[6108] := 16#8D59;
   // UNI[6109] := 16#8D5A;
   // UNI[6110] := 16#8D5B;
   // UNI[6111] := 16#8D5C;
   // UNI[6112] := 16#8D5D;
   // UNI[6113] := 16#8D5E;
   // UNI[6114] := 16#8D60;
   // UNI[6115] := 16#8D61;
   // UNI[6116] := 16#8D62;
   // UNI[6117] := 16#8D63;
   // UNI[6118] := 16#8D64;
   // UNI[6119] := 16#8D66;
   // UNI[6120] := 16#8D67;
   // UNI[6121] := 16#8D6B;
   // UNI[6122] := 16#8D6D;
   // UNI[6123] := 16#8D70;
   // UNI[6124] := 16#8D73;
   // UNI[6125] := 16#8D74;
   // UNI[6126] := 16#8D75;
   // UNI[6127] := 16#8D76;
   // UNI[6128] := 16#8D77;
   // UNI[6129] := 16#8D81;
   // UNI[6130] := 16#8D84;
   // UNI[6131] := 16#8D85;
   // UNI[6132] := 16#8D8A;
   // UNI[6133] := 16#8D8B;
   // UNI[6134] := 16#8D91;
   // UNI[6135] := 16#8D94;
   // UNI[6136] := 16#8D9F;
   // UNI[6137] := 16#8DA3;
   // UNI[6138] := 16#8DB1;
   // UNI[6139] := 16#8DB3;
   // UNI[6140] := 16#8DB4;
   // UNI[6141] := 16#8DB5;
   // UNI[6142] := 16#8DB8;
   // UNI[6143] := 16#8DBA;
   // UNI[6144] := 16#8DBC;
   // UNI[6145] := 16#8DBE;
   // UNI[6146] := 16#8DBF;
   // UNI[6147] := 16#8DC3;
   // UNI[6148] := 16#8DC4;
   // UNI[6149] := 16#8DC6;
   // UNI[6150] := 16#8DCB;
   // UNI[6151] := 16#8DCC;
   // UNI[6152] := 16#8DCE;
   // UNI[6153] := 16#8DCF;
   // UNI[6154] := 16#8DD1;
   // UNI[6155] := 16#8DD6;
   // UNI[6156] := 16#8DD7;
   // UNI[6157] := 16#8DDA;
   // UNI[6158] := 16#8DDB;
   // UNI[6159] := 16#8DDD;
   // UNI[6160] := 16#8DDE;
   // UNI[6161] := 16#8DDF;
   // UNI[6162] := 16#8DE3;
   // UNI[6163] := 16#8DE4;
   // UNI[6164] := 16#8DE8;
   // UNI[6165] := 16#8DEA;
   // UNI[6166] := 16#8DEB;
   // UNI[6167] := 16#8DEC;
   // UNI[6168] := 16#8DEF;
   // UNI[6169] := 16#8DF3;
   // UNI[6170] := 16#8DF5;
   // UNI[6171] := 16#8DF7;
   // UNI[6172] := 16#8DF8;
   // UNI[6173] := 16#8DF9;
   // UNI[6174] := 16#8DFA;
   // UNI[6175] := 16#8DFB;
   // UNI[6176] := 16#8DFD;
   // UNI[6177] := 16#8E05;
   // UNI[6178] := 16#8E09;
   // UNI[6179] := 16#8E0A;
   // UNI[6180] := 16#8E0C;
   // UNI[6181] := 16#8E0F;
   // UNI[6182] := 16#8E14;
   // UNI[6183] := 16#8E1D;
   // UNI[6184] := 16#8E1E;
   // UNI[6185] := 16#8E1F;
   // UNI[6186] := 16#8E22;
   // UNI[6187] := 16#8E23;
   // UNI[6188] := 16#8E29;
   // UNI[6189] := 16#8E2A;
   // UNI[6190] := 16#8E2C;
   // UNI[6191] := 16#8E2E;
   // UNI[6192] := 16#8E2F;
   // UNI[6193] := 16#8E31;
   // UNI[6194] := 16#8E35;
   // UNI[6195] := 16#8E39;
   // UNI[6196] := 16#8E3A;
   // UNI[6197] := 16#8E3D;
   // UNI[6198] := 16#8E40;
   // UNI[6199] := 16#8E41;
   // UNI[6200] := 16#8E42;
   // UNI[6201] := 16#8E44;
   // UNI[6202] := 16#8E47;
   // UNI[6203] := 16#8E48;
   // UNI[6204] := 16#8E49;
   // UNI[6205] := 16#8E4A;
   // UNI[6206] := 16#8E4B;
   // UNI[6207] := 16#8E51;
   // UNI[6208] := 16#8E52;
   // UNI[6209] := 16#8E59;
   // UNI[6210] := 16#8E66;
   // UNI[6211] := 16#8E69;
   // UNI[6212] := 16#8E6C;
   // UNI[6213] := 16#8E6D;
   // UNI[6214] := 16#8E6F;
   // UNI[6215] := 16#8E70;
   // UNI[6216] := 16#8E72;
   // UNI[6217] := 16#8E74;
   // UNI[6218] := 16#8E76;
   // UNI[6219] := 16#8E7C;
   // UNI[6220] := 16#8E7F;
   // UNI[6221] := 16#8E81;
   // UNI[6222] := 16#8E85;
   // UNI[6223] := 16#8E87;
   // UNI[6224] := 16#8E8F;
   // UNI[6225] := 16#8E90;
   // UNI[6226] := 16#8E94;
   // UNI[6227] := 16#8E9C;
   // UNI[6228] := 16#8E9E;
   // UNI[6229] := 16#8EAB;
   // UNI[6230] := 16#8EAC;
   // UNI[6231] := 16#8EAF;
   // UNI[6232] := 16#8EB2;
   // UNI[6233] := 16#8EBA;
   // UNI[6234] := 16#8ECE;
   // UNI[6235] := 16#8F66;
   // UNI[6236] := 16#8F67;
   // UNI[6237] := 16#8F68;
   // UNI[6238] := 16#8F69;
   // UNI[6239] := 16#8F6B;
   // UNI[6240] := 16#8F6C;
   // UNI[6241] := 16#8F6D;
   // UNI[6242] := 16#8F6E;
   // UNI[6243] := 16#8F6F;
   // UNI[6244] := 16#8F70;
   // UNI[6245] := 16#8F71;
   // UNI[6246] := 16#8F72;
   // UNI[6247] := 16#8F73;
   // UNI[6248] := 16#8F74;
   // UNI[6249] := 16#8F75;
   // UNI[6250] := 16#8F76;
   // UNI[6251] := 16#8F77;
   // UNI[6252] := 16#8F78;
   // UNI[6253] := 16#8F79;
   // UNI[6254] := 16#8F7A;
   // UNI[6255] := 16#8F7B;
   // UNI[6256] := 16#8F7C;
   // UNI[6257] := 16#8F7D;
   // UNI[6258] := 16#8F7E;
   // UNI[6259] := 16#8F7F;
   // UNI[6260] := 16#8F81;
   // UNI[6261] := 16#8F82;
   // UNI[6262] := 16#8F83;
   // UNI[6263] := 16#8F84;
   // UNI[6264] := 16#8F85;
   // UNI[6265] := 16#8F86;
   // UNI[6266] := 16#8F87;
   // UNI[6267] := 16#8F88;
   // UNI[6268] := 16#8F89;
   // UNI[6269] := 16#8F8A;
   // UNI[6270] := 16#8F8B;
   // UNI[6271] := 16#8F8D;
   // UNI[6272] := 16#8F8E;
   // UNI[6273] := 16#8F8F;
   // UNI[6274] := 16#8F90;
   // UNI[6275] := 16#8F91;
   // UNI[6276] := 16#8F93;
   // UNI[6277] := 16#8F94;
   // UNI[6278] := 16#8F95;
   // UNI[6279] := 16#8F96;
   // UNI[6280] := 16#8F97;
   // UNI[6281] := 16#8F98;
   // UNI[6282] := 16#8F99;
   // UNI[6283] := 16#8F9A;
   // UNI[6284] := 16#8F9B;
   // UNI[6285] := 16#8F9C;
   // UNI[6286] := 16#8F9E;
   // UNI[6287] := 16#8F9F;
   // UNI[6288] := 16#8FA3;
   // UNI[6289] := 16#8FA8;
   // UNI[6290] := 16#8FA9;
   // UNI[6291] := 16#8FAB;
   // UNI[6292] := 16#8FB0;
   // UNI[6293] := 16#8FB1;
   // UNI[6294] := 16#8FB6;
   // UNI[6295] := 16#8FB9;
   // UNI[6296] := 16#8FBD;
   // UNI[6297] := 16#8FBE;
   // UNI[6298] := 16#8FC1;
   // UNI[6299] := 16#8FC2;
   // UNI[6300] := 16#8FC4;
   // UNI[6301] := 16#8FC5;
   // UNI[6302] := 16#8FC7;
   // UNI[6303] := 16#8FC8;
   // UNI[6304] := 16#8FCE;
   // UNI[6305] := 16#8FD0;
   // UNI[6306] := 16#8FD1;
   // UNI[6307] := 16#8FD3;
   // UNI[6308] := 16#8FD4;
   // UNI[6309] := 16#8FD5;
   // UNI[6310] := 16#8FD8;
   // UNI[6311] := 16#8FD9;
   // UNI[6312] := 16#8FDB;
   // UNI[6313] := 16#8FDC;
   // UNI[6314] := 16#8FDD;
   // UNI[6315] := 16#8FDE;
   // UNI[6316] := 16#8FDF;
   // UNI[6317] := 16#8FE2;
   // UNI[6318] := 16#8FE4;
   // UNI[6319] := 16#8FE5;
   // UNI[6320] := 16#8FE6;
   // UNI[6321] := 16#8FE8;
   // UNI[6322] := 16#8FE9;
   // UNI[6323] := 16#8FEA;
   // UNI[6324] := 16#8FEB;
   // UNI[6325] := 16#8FED;
   // UNI[6326] := 16#8FEE;
   // UNI[6327] := 16#8FF0;
   // UNI[6328] := 16#8FF3;
   // UNI[6329] := 16#8FF7;
   // UNI[6330] := 16#8FF8;
   // UNI[6331] := 16#8FF9;
   // UNI[6332] := 16#8FFD;
   // UNI[6333] := 16#9000;
   // UNI[6334] := 16#9001;
   // UNI[6335] := 16#9002;
   // UNI[6336] := 16#9003;
   // UNI[6337] := 16#9004;
   // UNI[6338] := 16#9005;
   // UNI[6339] := 16#9006;
   // UNI[6340] := 16#9009;
   // UNI[6341] := 16#900A;
   // UNI[6342] := 16#900B;
   // UNI[6343] := 16#900D;
   // UNI[6344] := 16#900F;
   // UNI[6345] := 16#9010;
   // UNI[6346] := 16#9011;
   // UNI[6347] := 16#9012;
   // UNI[6348] := 16#9014;
   // UNI[6349] := 16#9016;
   // UNI[6350] := 16#9017;
   // UNI[6351] := 16#901A;
   // UNI[6352] := 16#901B;
   // UNI[6353] := 16#901D;
   // UNI[6354] := 16#901E;
   // UNI[6355] := 16#901F;
   // UNI[6356] := 16#9020;
   // UNI[6357] := 16#9021;
   // UNI[6358] := 16#9022;
   // UNI[6359] := 16#9026;
   // UNI[6360] := 16#902D;
   // UNI[6361] := 16#902E;
   // UNI[6362] := 16#902F;
   // UNI[6363] := 16#9035;
   // UNI[6364] := 16#9036;
   // UNI[6365] := 16#9038;
   // UNI[6366] := 16#903B;
   // UNI[6367] := 16#903C;
   // UNI[6368] := 16#903E;
   // UNI[6369] := 16#9041;
   // UNI[6370] := 16#9042;
   // UNI[6371] := 16#9044;
   // UNI[6372] := 16#9047;
   // UNI[6373] := 16#904D;
   // UNI[6374] := 16#904F;
   // UNI[6375] := 16#9050;
   // UNI[6376] := 16#9051;
   // UNI[6377] := 16#9052;
   // UNI[6378] := 16#9053;
   // UNI[6379] := 16#9057;
   // UNI[6380] := 16#9058;
   // UNI[6381] := 16#905B;
   // UNI[6382] := 16#9062;
   // UNI[6383] := 16#9063;
   // UNI[6384] := 16#9065;
   // UNI[6385] := 16#9068;
   // UNI[6386] := 16#906D;
   // UNI[6387] := 16#906E;
   // UNI[6388] := 16#9074;
   // UNI[6389] := 16#9075;
   // UNI[6390] := 16#907D;
   // UNI[6391] := 16#907F;
   // UNI[6392] := 16#9080;
   // UNI[6393] := 16#9082;
   // UNI[6394] := 16#9083;
   // UNI[6395] := 16#9088;
   // UNI[6396] := 16#908B;
   // UNI[6397] := 16#9091;
   // UNI[6398] := 16#9093;
   // UNI[6399] := 16#9095;
   // UNI[6400] := 16#9097;
   // UNI[6401] := 16#9099;
   // UNI[6402] := 16#909B;
   // UNI[6403] := 16#909D;
   // UNI[6404] := 16#90A1;
   // UNI[6405] := 16#90A2;
   // UNI[6406] := 16#90A3;
   // UNI[6407] := 16#90A6;
   // UNI[6408] := 16#90AA;
   // UNI[6409] := 16#90AC;
   // UNI[6410] := 16#90AE;
   // UNI[6411] := 16#90AF;
   // UNI[6412] := 16#90B0;
   // UNI[6413] := 16#90B1;
   // UNI[6414] := 16#90B3;
   // UNI[6415] := 16#90B4;
   // UNI[6416] := 16#90B5;
   // UNI[6417] := 16#90B6;
   // UNI[6418] := 16#90B8;
   // UNI[6419] := 16#90B9;
   // UNI[6420] := 16#90BA;
   // UNI[6421] := 16#90BB;
   // UNI[6422] := 16#90BE;
   // UNI[6423] := 16#90C1;
   // UNI[6424] := 16#90C4;
   // UNI[6425] := 16#90C5;
   // UNI[6426] := 16#90C7;
   // UNI[6427] := 16#90CA;
   // UNI[6428] := 16#90CE;
   // UNI[6429] := 16#90CF;
   // UNI[6430] := 16#90D0;
   // UNI[6431] := 16#90D1;
   // UNI[6432] := 16#90D3;
   // UNI[6433] := 16#90D7;
   // UNI[6434] := 16#90DB;
   // UNI[6435] := 16#90DC;
   // UNI[6436] := 16#90DD;
   // UNI[6437] := 16#90E1;
   // UNI[6438] := 16#90E2;
   // UNI[6439] := 16#90E6;
   // UNI[6440] := 16#90E7;
   // UNI[6441] := 16#90E8;
   // UNI[6442] := 16#90EB;
   // UNI[6443] := 16#90ED;
   // UNI[6444] := 16#90EF;
   // UNI[6445] := 16#90F4;
   // UNI[6446] := 16#90F8;
   // UNI[6447] := 16#90FD;
   // UNI[6448] := 16#90FE;
   // UNI[6449] := 16#9102;
   // UNI[6450] := 16#9104;
   // UNI[6451] := 16#9119;
   // UNI[6452] := 16#911E;
   // UNI[6453] := 16#9122;
   // UNI[6454] := 16#9123;
   // UNI[6455] := 16#912F;
   // UNI[6456] := 16#9131;
   // UNI[6457] := 16#9139;
   // UNI[6458] := 16#9143;
   // UNI[6459] := 16#9146;
   // UNI[6460] := 16#9149;
   // UNI[6461] := 16#914A;
   // UNI[6462] := 16#914B;
   // UNI[6463] := 16#914C;
   // UNI[6464] := 16#914D;
   // UNI[6465] := 16#914E;
   // UNI[6466] := 16#914F;
   // UNI[6467] := 16#9150;
   // UNI[6468] := 16#9152;
   // UNI[6469] := 16#9157;
   // UNI[6470] := 16#915A;
   // UNI[6471] := 16#915D;
   // UNI[6472] := 16#915E;
   // UNI[6473] := 16#9161;
   // UNI[6474] := 16#9162;
   // UNI[6475] := 16#9163;
   // UNI[6476] := 16#9164;
   // UNI[6477] := 16#9165;
   // UNI[6478] := 16#9169;
   // UNI[6479] := 16#916A;
   // UNI[6480] := 16#916C;
   // UNI[6481] := 16#916E;
   // UNI[6482] := 16#916F;
   // UNI[6483] := 16#9170;
   // UNI[6484] := 16#9171;
   // UNI[6485] := 16#9172;
   // UNI[6486] := 16#9174;
   // UNI[6487] := 16#9175;
   // UNI[6488] := 16#9176;
   // UNI[6489] := 16#9177;
   // UNI[6490] := 16#9178;
   // UNI[6491] := 16#9179;
   // UNI[6492] := 16#917D;
   // UNI[6493] := 16#917E;
   // UNI[6494] := 16#917F;
   // UNI[6495] := 16#9185;
   // UNI[6496] := 16#9187;
   // UNI[6497] := 16#9189;
   // UNI[6498] := 16#918B;
   // UNI[6499] := 16#918C;
   // UNI[6500] := 16#918D;
   // UNI[6501] := 16#9190;
   // UNI[6502] := 16#9191;
   // UNI[6503] := 16#9192;
   // UNI[6504] := 16#919A;
   // UNI[6505] := 16#919B;
   // UNI[6506] := 16#91A2;
   // UNI[6507] := 16#91A3;
   // UNI[6508] := 16#91AA;
   // UNI[6509] := 16#91AD;
   // UNI[6510] := 16#91AE;
   // UNI[6511] := 16#91AF;
   // UNI[6512] := 16#91B4;
   // UNI[6513] := 16#91B5;
   // UNI[6514] := 16#91BA;
   // UNI[6515] := 16#91C7;
   // UNI[6516] := 16#91C9;
   // UNI[6517] := 16#91CA;
   // UNI[6518] := 16#91CC;
   // UNI[6519] := 16#91CD;
   // UNI[6520] := 16#91CE;
   // UNI[6521] := 16#91CF;
   // UNI[6522] := 16#91D1;
   // UNI[6523] := 16#91DC;
   // UNI[6524] := 16#9274;
   // UNI[6525] := 16#928E;
   // UNI[6526] := 16#92AE;
   // UNI[6527] := 16#92C8;
   // UNI[6528] := 16#933E;
   // UNI[6529] := 16#936A;
   // UNI[6530] := 16#938F;
   // UNI[6531] := 16#93CA;
   // UNI[6532] := 16#93D6;
   // UNI[6533] := 16#943E;
   // UNI[6534] := 16#946B;
   // UNI[6535] := 16#9485;
   // UNI[6536] := 16#9486;
   // UNI[6537] := 16#9487;
   // UNI[6538] := 16#9488;
   // UNI[6539] := 16#9489;
   // UNI[6540] := 16#948A;
   // UNI[6541] := 16#948B;
   // UNI[6542] := 16#948C;
   // UNI[6543] := 16#948D;
   // UNI[6544] := 16#948E;
   // UNI[6545] := 16#948F;
   // UNI[6546] := 16#9490;
   // UNI[6547] := 16#9492;
   // UNI[6548] := 16#9493;
   // UNI[6549] := 16#9494;
   // UNI[6550] := 16#9495;
   // UNI[6551] := 16#9497;
   // UNI[6552] := 16#9499;
   // UNI[6553] := 16#949A;
   // UNI[6554] := 16#949B;
   // UNI[6555] := 16#949C;
   // UNI[6556] := 16#949D;
   // UNI[6557] := 16#949E;
   // UNI[6558] := 16#949F;
   // UNI[6559] := 16#94A0;
   // UNI[6560] := 16#94A1;
   // UNI[6561] := 16#94A2;
   // UNI[6562] := 16#94A3;
   // UNI[6563] := 16#94A4;
   // UNI[6564] := 16#94A5;
   // UNI[6565] := 16#94A6;
   // UNI[6566] := 16#94A7;
   // UNI[6567] := 16#94A8;
   // UNI[6568] := 16#94A9;
   // UNI[6569] := 16#94AA;
   // UNI[6570] := 16#94AB;
   // UNI[6571] := 16#94AC;
   // UNI[6572] := 16#94AD;
   // UNI[6573] := 16#94AE;
   // UNI[6574] := 16#94AF;
   // UNI[6575] := 16#94B0;
   // UNI[6576] := 16#94B1;
   // UNI[6577] := 16#94B2;
   // UNI[6578] := 16#94B3;
   // UNI[6579] := 16#94B4;
   // UNI[6580] := 16#94B5;
   // UNI[6581] := 16#94B6;
   // UNI[6582] := 16#94B7;
   // UNI[6583] := 16#94B8;
   // UNI[6584] := 16#94B9;
   // UNI[6585] := 16#94BA;
   // UNI[6586] := 16#94BB;
   // UNI[6587] := 16#94BC;
   // UNI[6588] := 16#94BD;
   // UNI[6589] := 16#94BE;
   // UNI[6590] := 16#94BF;
   // UNI[6591] := 16#94C0;
   // UNI[6592] := 16#94C1;
   // UNI[6593] := 16#94C2;
   // UNI[6594] := 16#94C3;
   // UNI[6595] := 16#94C4;
   // UNI[6596] := 16#94C5;
   // UNI[6597] := 16#94C6;
   // UNI[6598] := 16#94C8;
   // UNI[6599] := 16#94C9;
   // UNI[6600] := 16#94CA;
   // UNI[6601] := 16#94CB;
   // UNI[6602] := 16#94CC;
   // UNI[6603] := 16#94CD;
   // UNI[6604] := 16#94CE;
   // UNI[6605] := 16#94D0;
   // UNI[6606] := 16#94D1;
   // UNI[6607] := 16#94D2;
   // UNI[6608] := 16#94D5;
   // UNI[6609] := 16#94D6;
   // UNI[6610] := 16#94D7;
   // UNI[6611] := 16#94D8;
   // UNI[6612] := 16#94D9;
   // UNI[6613] := 16#94DB;
   // UNI[6614] := 16#94DC;
   // UNI[6615] := 16#94DD;
   // UNI[6616] := 16#94DE;
   // UNI[6617] := 16#94DF;
   // UNI[6618] := 16#94E0;
   // UNI[6619] := 16#94E1;
   // UNI[6620] := 16#94E2;
   // UNI[6621] := 16#94E3;
   // UNI[6622] := 16#94E4;
   // UNI[6623] := 16#94E5;
   // UNI[6624] := 16#94E7;
   // UNI[6625] := 16#94E8;
   // UNI[6626] := 16#94E9;
   // UNI[6627] := 16#94EA;
   // UNI[6628] := 16#94EB;
   // UNI[6629] := 16#94EC;
   // UNI[6630] := 16#94ED;
   // UNI[6631] := 16#94EE;
   // UNI[6632] := 16#94EF;
   // UNI[6633] := 16#94F0;
   // UNI[6634] := 16#94F1;
   // UNI[6635] := 16#94F2;
   // UNI[6636] := 16#94F3;
   // UNI[6637] := 16#94F4;
   // UNI[6638] := 16#94F5;
   // UNI[6639] := 16#94F6;
   // UNI[6640] := 16#94F7;
   // UNI[6641] := 16#94F8;
   // UNI[6642] := 16#94F9;
   // UNI[6643] := 16#94FA;
   // UNI[6644] := 16#94FC;
   // UNI[6645] := 16#94FD;
   // UNI[6646] := 16#94FE;
   // UNI[6647] := 16#94FF;
   // UNI[6648] := 16#9500;
   // UNI[6649] := 16#9501;
   // UNI[6650] := 16#9502;
   // UNI[6651] := 16#9503;
   // UNI[6652] := 16#9504;
   // UNI[6653] := 16#9505;
   // UNI[6654] := 16#9506;
   // UNI[6655] := 16#9507;
   // UNI[6656] := 16#9508;
   // UNI[6657] := 16#9509;
   // UNI[6658] := 16#950A;
   // UNI[6659] := 16#950B;
   // UNI[6660] := 16#950C;
   // UNI[6661] := 16#950D;
   // UNI[6662] := 16#950E;
   // UNI[6663] := 16#950F;
   // UNI[6664] := 16#9510;
   // UNI[6665] := 16#9511;
   // UNI[6666] := 16#9512;
   // UNI[6667] := 16#9513;
   // UNI[6668] := 16#9514;
   // UNI[6669] := 16#9515;
   // UNI[6670] := 16#9516;
   // UNI[6671] := 16#9517;
   // UNI[6672] := 16#9518;
   // UNI[6673] := 16#9519;
   // UNI[6674] := 16#951A;
   // UNI[6675] := 16#951B;
   // UNI[6676] := 16#951D;
   // UNI[6677] := 16#951E;
   // UNI[6678] := 16#951F;
   // UNI[6679] := 16#9521;
   // UNI[6680] := 16#9522;
   // UNI[6681] := 16#9523;
   // UNI[6682] := 16#9524;
   // UNI[6683] := 16#9525;
   // UNI[6684] := 16#9526;
   // UNI[6685] := 16#9528;
   // UNI[6686] := 16#9529;
   // UNI[6687] := 16#952A;
   // UNI[6688] := 16#952B;
   // UNI[6689] := 16#952C;
   // UNI[6690] := 16#952D;
   // UNI[6691] := 16#952E;
   // UNI[6692] := 16#952F;
   // UNI[6693] := 16#9530;
   // UNI[6694] := 16#9531;
   // UNI[6695] := 16#9532;
   // UNI[6696] := 16#9534;
   // UNI[6697] := 16#9535;
   // UNI[6698] := 16#9536;
   // UNI[6699] := 16#9537;
   // UNI[6700] := 16#9538;
   // UNI[6701] := 16#9539;
   // UNI[6702] := 16#953A;
   // UNI[6703] := 16#953B;
   // UNI[6704] := 16#953C;
   // UNI[6705] := 16#953E;
   // UNI[6706] := 16#953F;
   // UNI[6707] := 16#9540;
   // UNI[6708] := 16#9541;
   // UNI[6709] := 16#9542;
   // UNI[6710] := 16#9544;
   // UNI[6711] := 16#9545;
   // UNI[6712] := 16#9546;
   // UNI[6713] := 16#9547;
   // UNI[6714] := 16#9549;
   // UNI[6715] := 16#954A;
   // UNI[6716] := 16#954C;
   // UNI[6717] := 16#954D;
   // UNI[6718] := 16#954E;
   // UNI[6719] := 16#954F;
   // UNI[6720] := 16#9550;
   // UNI[6721] := 16#9551;
   // UNI[6722] := 16#9552;
   // UNI[6723] := 16#9553;
   // UNI[6724] := 16#9554;
   // UNI[6725] := 16#9556;
   // UNI[6726] := 16#9557;
   // UNI[6727] := 16#9558;
   // UNI[6728] := 16#9559;
   // UNI[6729] := 16#955B;
   // UNI[6730] := 16#955C;
   // UNI[6731] := 16#955D;
   // UNI[6732] := 16#955E;
   // UNI[6733] := 16#955F;
   // UNI[6734] := 16#9561;
   // UNI[6735] := 16#9562;
   // UNI[6736] := 16#9563;
   // UNI[6737] := 16#9564;
   // UNI[6738] := 16#9565;
   // UNI[6739] := 16#9566;
   // UNI[6740] := 16#9567;
   // UNI[6741] := 16#9568;
   // UNI[6742] := 16#9569;
   // UNI[6743] := 16#956A;
   // UNI[6744] := 16#956B;
   // UNI[6745] := 16#956C;
   // UNI[6746] := 16#956D;
   // UNI[6747] := 16#956F;
   // UNI[6748] := 16#9570;
   // UNI[6749] := 16#9571;
   // UNI[6750] := 16#9572;
   // UNI[6751] := 16#9573;
   // UNI[6752] := 16#9576;
   // UNI[6753] := 16#957F;
   // UNI[6754] := 16#95E8;
   // UNI[6755] := 16#95E9;
   // UNI[6756] := 16#95EA;
   // UNI[6757] := 16#95EB;
   // UNI[6758] := 16#95ED;
   // UNI[6759] := 16#95EE;
   // UNI[6760] := 16#95EF;
   // UNI[6761] := 16#95F0;
   // UNI[6762] := 16#95F1;
   // UNI[6763] := 16#95F2;
   // UNI[6764] := 16#95F3;
   // UNI[6765] := 16#95F4;
   // UNI[6766] := 16#95F5;
   // UNI[6767] := 16#95F6;
   // UNI[6768] := 16#95F7;
   // UNI[6769] := 16#95F8;
   // UNI[6770] := 16#95F9;
   // UNI[6771] := 16#95FA;
   // UNI[6772] := 16#95FB;
   // UNI[6773] := 16#95FC;
   // UNI[6774] := 16#95FD;
   // UNI[6775] := 16#95FE;
   // UNI[6776] := 16#9600;
   // UNI[6777] := 16#9601;
   // UNI[6778] := 16#9602;
   // UNI[6779] := 16#9603;
   // UNI[6780] := 16#9604;
   // UNI[6781] := 16#9605;
   // UNI[6782] := 16#9606;
   // UNI[6783] := 16#9608;
   // UNI[6784] := 16#9609;
   // UNI[6785] := 16#960A;
   // UNI[6786] := 16#960B;
   // UNI[6787] := 16#960C;
   // UNI[6788] := 16#960D;
   // UNI[6789] := 16#960E;
   // UNI[6790] := 16#960F;
   // UNI[6791] := 16#9610;
   // UNI[6792] := 16#9611;
   // UNI[6793] := 16#9612;
   // UNI[6794] := 16#9614;
   // UNI[6795] := 16#9615;
   // UNI[6796] := 16#9616;
   // UNI[6797] := 16#9617;
   // UNI[6798] := 16#9619;
   // UNI[6799] := 16#961A;
   // UNI[6800] := 16#961C;
   // UNI[6801] := 16#961D;
   // UNI[6802] := 16#961F;
   // UNI[6803] := 16#9621;
   // UNI[6804] := 16#9622;
   // UNI[6805] := 16#962A;
   // UNI[6806] := 16#962E;
   // UNI[6807] := 16#9631;
   // UNI[6808] := 16#9632;
   // UNI[6809] := 16#9633;
   // UNI[6810] := 16#9634;
   // UNI[6811] := 16#9635;
   // UNI[6812] := 16#9636;
   // UNI[6813] := 16#963B;
   // UNI[6814] := 16#963C;
   // UNI[6815] := 16#963D;
   // UNI[6816] := 16#963F;
   // UNI[6817] := 16#9640;
   // UNI[6818] := 16#9642;
   // UNI[6819] := 16#9644;
   // UNI[6820] := 16#9645;
   // UNI[6821] := 16#9646;
   // UNI[6822] := 16#9647;
   // UNI[6823] := 16#9648;
   // UNI[6824] := 16#9649;
   // UNI[6825] := 16#964B;
   // UNI[6826] := 16#964C;
   // UNI[6827] := 16#964D;
   // UNI[6828] := 16#9650;
   // UNI[6829] := 16#9654;
   // UNI[6830] := 16#9655;
   // UNI[6831] := 16#965B;
   // UNI[6832] := 16#965F;
   // UNI[6833] := 16#9661;
   // UNI[6834] := 16#9662;
   // UNI[6835] := 16#9664;
   // UNI[6836] := 16#9667;
   // UNI[6837] := 16#9668;
   // UNI[6838] := 16#9669;
   // UNI[6839] := 16#966A;
   // UNI[6840] := 16#966C;
   // UNI[6841] := 16#9672;
   // UNI[6842] := 16#9674;
   // UNI[6843] := 16#9675;
   // UNI[6844] := 16#9676;
   // UNI[6845] := 16#9677;
   // UNI[6846] := 16#9685;
   // UNI[6847] := 16#9686;
   // UNI[6848] := 16#9688;
   // UNI[6849] := 16#968B;
   // UNI[6850] := 16#968D;
   // UNI[6851] := 16#968F;
   // UNI[6852] := 16#9690;
   // UNI[6853] := 16#9694;
   // UNI[6854] := 16#9697;
   // UNI[6855] := 16#9698;
   // UNI[6856] := 16#9699;
   // UNI[6857] := 16#969C;
   // UNI[6858] := 16#96A7;
   // UNI[6859] := 16#96B0;
   // UNI[6860] := 16#96B3;
   // UNI[6861] := 16#96B6;
   // UNI[6862] := 16#96B9;
   // UNI[6863] := 16#96BC;
   // UNI[6864] := 16#96BD;
   // UNI[6865] := 16#96BE;
   // UNI[6866] := 16#96C0;
   // UNI[6867] := 16#96C1;
   // UNI[6868] := 16#96C4;
   // UNI[6869] := 16#96C5;
   // UNI[6870] := 16#96C6;
   // UNI[6871] := 16#96C7;
   // UNI[6872] := 16#96C9;
   // UNI[6873] := 16#96CC;
   // UNI[6874] := 16#96CD;
   // UNI[6875] := 16#96CE;
   // UNI[6876] := 16#96CF;
   // UNI[6877] := 16#96D2;
   // UNI[6878] := 16#96D5;
   // UNI[6879] := 16#96E0;
   // UNI[6880] := 16#96E8;
   // UNI[6881] := 16#96E9;
   // UNI[6882] := 16#96EA;
   // UNI[6883] := 16#96EF;
   // UNI[6884] := 16#96F3;
   // UNI[6885] := 16#96F6;
   // UNI[6886] := 16#96F7;
   // UNI[6887] := 16#96F9;
   // UNI[6888] := 16#96FE;
   // UNI[6889] := 16#9700;
   // UNI[6890] := 16#9701;
   // UNI[6891] := 16#9704;
   // UNI[6892] := 16#9706;
   // UNI[6893] := 16#9707;
   // UNI[6894] := 16#9708;
   // UNI[6895] := 16#9709;
   // UNI[6896] := 16#970D;
   // UNI[6897] := 16#970E;
   // UNI[6898] := 16#970F;
   // UNI[6899] := 16#9713;
   // UNI[6900] := 16#9716;
   // UNI[6901] := 16#971C;
   // UNI[6902] := 16#971E;
   // UNI[6903] := 16#972A;
   // UNI[6904] := 16#972D;
   // UNI[6905] := 16#9730;
   // UNI[6906] := 16#9732;
   // UNI[6907] := 16#9738;
   // UNI[6908] := 16#9739;
   // UNI[6909] := 16#973E;
   // UNI[6910] := 16#9752;
   // UNI[6911] := 16#9753;
   // UNI[6912] := 16#9756;
   // UNI[6913] := 16#9759;
   // UNI[6914] := 16#975B;
   // UNI[6915] := 16#975E;
   // UNI[6916] := 16#9760;
   // UNI[6917] := 16#9761;
   // UNI[6918] := 16#9762;
   // UNI[6919] := 16#9765;
   // UNI[6920] := 16#9769;
   // UNI[6921] := 16#9773;
   // UNI[6922] := 16#9774;
   // UNI[6923] := 16#9776;
   // UNI[6924] := 16#977C;
   // UNI[6925] := 16#9785;
   // UNI[6926] := 16#978B;
   // UNI[6927] := 16#978D;
   // UNI[6928] := 16#9791;
   // UNI[6929] := 16#9792;
   // UNI[6930] := 16#9794;
   // UNI[6931] := 16#9798;
   // UNI[6932] := 16#97A0;
   // UNI[6933] := 16#97A3;
   // UNI[6934] := 16#97AB;
   // UNI[6935] := 16#97AD;
   // UNI[6936] := 16#97AF;
   // UNI[6937] := 16#97B2;
   // UNI[6938] := 16#97B4;
   // UNI[6939] := 16#97E6;
   // UNI[6940] := 16#97E7;
   // UNI[6941] := 16#97E9;
   // UNI[6942] := 16#97EA;
   // UNI[6943] := 16#97EB;
   // UNI[6944] := 16#97EC;
   // UNI[6945] := 16#97ED;
   // UNI[6946] := 16#97F3;
   // UNI[6947] := 16#97F5;
   // UNI[6948] := 16#97F6;
   // UNI[6949] := 16#9875;
   // UNI[6950] := 16#9876;
   // UNI[6951] := 16#9877;
   // UNI[6952] := 16#9878;
   // UNI[6953] := 16#9879;
   // UNI[6954] := 16#987A;
   // UNI[6955] := 16#987B;
   // UNI[6956] := 16#987C;
   // UNI[6957] := 16#987D;
   // UNI[6958] := 16#987E;
   // UNI[6959] := 16#987F;
   // UNI[6960] := 16#9880;
   // UNI[6961] := 16#9881;
   // UNI[6962] := 16#9882;
   // UNI[6963] := 16#9883;
   // UNI[6964] := 16#9884;
   // UNI[6965] := 16#9885;
   // UNI[6966] := 16#9886;
   // UNI[6967] := 16#9887;
   // UNI[6968] := 16#9888;
   // UNI[6969] := 16#9889;
   // UNI[6970] := 16#988A;
   // UNI[6971] := 16#988C;
   // UNI[6972] := 16#988D;
   // UNI[6973] := 16#988F;
   // UNI[6974] := 16#9890;
   // UNI[6975] := 16#9891;
   // UNI[6976] := 16#9893;
   // UNI[6977] := 16#9894;
   // UNI[6978] := 16#9896;
   // UNI[6979] := 16#9897;
   // UNI[6980] := 16#9898;
   // UNI[6981] := 16#989A;
   // UNI[6982] := 16#989B;
   // UNI[6983] := 16#989C;
   // UNI[6984] := 16#989D;
   // UNI[6985] := 16#989E;
   // UNI[6986] := 16#989F;
   // UNI[6987] := 16#98A0;
   // UNI[6988] := 16#98A1;
   // UNI[6989] := 16#98A2;
   // UNI[6990] := 16#98A4;
   // UNI[6991] := 16#98A5;
   // UNI[6992] := 16#98A6;
   // UNI[6993] := 16#98A7;
   // UNI[6994] := 16#98CE;
   // UNI[6995] := 16#98D1;
   // UNI[6996] := 16#98D2;
   // UNI[6997] := 16#98D3;
   // UNI[6998] := 16#98D5;
   // UNI[6999] := 16#98D8;
   // UNI[7000] := 16#98D9;
   // UNI[7001] := 16#98DA;
   // UNI[7002] := 16#98DE;
   // UNI[7003] := 16#98DF;
   // UNI[7004] := 16#98E7;
   // UNI[7005] := 16#98E8;
   // UNI[7006] := 16#990D;
   // UNI[7007] := 16#9910;
   // UNI[7008] := 16#992E;
   // UNI[7009] := 16#9954;
   // UNI[7010] := 16#9955;
   // UNI[7011] := 16#9963;
   // UNI[7012] := 16#9965;
   // UNI[7013] := 16#9967;
   // UNI[7014] := 16#9968;
   // UNI[7015] := 16#9969;
   // UNI[7016] := 16#996A;
   // UNI[7017] := 16#996B;
   // UNI[7018] := 16#996C;
   // UNI[7019] := 16#996D;
   // UNI[7020] := 16#996E;
   // UNI[7021] := 16#996F;
   // UNI[7022] := 16#9970;
   // UNI[7023] := 16#9971;
   // UNI[7024] := 16#9972;
   // UNI[7025] := 16#9974;
   // UNI[7026] := 16#9975;
   // UNI[7027] := 16#9976;
   // UNI[7028] := 16#9977;
   // UNI[7029] := 16#997A;
   // UNI[7030] := 16#997C;
   // UNI[7031] := 16#997D;
   // UNI[7032] := 16#997F;
   // UNI[7033] := 16#9980;
   // UNI[7034] := 16#9981;
   // UNI[7035] := 16#9984;
   // UNI[7036] := 16#9985;
   // UNI[7037] := 16#9986;
   // UNI[7038] := 16#9987;
   // UNI[7039] := 16#9988;
   // UNI[7040] := 16#998A;
   // UNI[7041] := 16#998B;
   // UNI[7042] := 16#998D;
   // UNI[7043] := 16#998F;
   // UNI[7044] := 16#9990;
   // UNI[7045] := 16#9991;
   // UNI[7046] := 16#9992;
   // UNI[7047] := 16#9993;
   // UNI[7048] := 16#9994;
   // UNI[7049] := 16#9995;
   // UNI[7050] := 16#9996;
   // UNI[7051] := 16#9997;
   // UNI[7052] := 16#9998;
   // UNI[7053] := 16#9999;
   // UNI[7054] := 16#99A5;
   // UNI[7055] := 16#99A8;
   // UNI[7056] := 16#9A6C;
   // UNI[7057] := 16#9A6D;
   // UNI[7058] := 16#9A6E;
   // UNI[7059] := 16#9A6F;
   // UNI[7060] := 16#9A70;
   // UNI[7061] := 16#9A71;
   // UNI[7062] := 16#9A73;
   // UNI[7063] := 16#9A74;
   // UNI[7064] := 16#9A75;
   // UNI[7065] := 16#9A76;
   // UNI[7066] := 16#9A77;
   // UNI[7067] := 16#9A78;
   // UNI[7068] := 16#9A79;
   // UNI[7069] := 16#9A7A;
   // UNI[7070] := 16#9A7B;
   // UNI[7071] := 16#9A7C;
   // UNI[7072] := 16#9A7D;
   // UNI[7073] := 16#9A7E;
   // UNI[7074] := 16#9A7F;
   // UNI[7075] := 16#9A80;
   // UNI[7076] := 16#9A81;
   // UNI[7077] := 16#9A82;
   // UNI[7078] := 16#9A84;
   // UNI[7079] := 16#9A85;
   // UNI[7080] := 16#9A86;
   // UNI[7081] := 16#9A87;
   // UNI[7082] := 16#9A88;
   // UNI[7083] := 16#9A8A;
   // UNI[7084] := 16#9A8B;
   // UNI[7085] := 16#9A8C;
   // UNI[7086] := 16#9A8F;
   // UNI[7087] := 16#9A90;
   // UNI[7088] := 16#9A91;
   // UNI[7089] := 16#9A92;
   // UNI[7090] := 16#9A93;
   // UNI[7091] := 16#9A96;
   // UNI[7092] := 16#9A97;
   // UNI[7093] := 16#9A98;
   // UNI[7094] := 16#9A9A;
   // UNI[7095] := 16#9A9B;
   // UNI[7096] := 16#9A9C;
   // UNI[7097] := 16#9A9D;
   // UNI[7098] := 16#9A9E;
   // UNI[7099] := 16#9A9F;
   // UNI[7100] := 16#9AA0;
   // UNI[7101] := 16#9AA1;
   // UNI[7102] := 16#9AA2;
   // UNI[7103] := 16#9AA3;
   // UNI[7104] := 16#9AA4;
   // UNI[7105] := 16#9AA5;
   // UNI[7106] := 16#9AA7;
   // UNI[7107] := 16#9AA8;
   // UNI[7108] := 16#9AB0;
   // UNI[7109] := 16#9AB1;
   // UNI[7110] := 16#9AB6;
   // UNI[7111] := 16#9AB7;
   // UNI[7112] := 16#9AB8;
   // UNI[7113] := 16#9ABA;
   // UNI[7114] := 16#9ABC;
   // UNI[7115] := 16#9AC0;
   // UNI[7116] := 16#9AC1;
   // UNI[7117] := 16#9AC2;
   // UNI[7118] := 16#9AC5;
   // UNI[7119] := 16#9ACB;
   // UNI[7120] := 16#9ACC;
   // UNI[7121] := 16#9AD1;
   // UNI[7122] := 16#9AD3;
   // UNI[7123] := 16#9AD8;
   // UNI[7124] := 16#9ADF;
   // UNI[7125] := 16#9AE1;
   // UNI[7126] := 16#9AE6;
   // UNI[7127] := 16#9AEB;
   // UNI[7128] := 16#9AED;
   // UNI[7129] := 16#9AEF;
   // UNI[7130] := 16#9AF9;
   // UNI[7131] := 16#9AFB;
   // UNI[7132] := 16#9B03;
   // UNI[7133] := 16#9B08;
   // UNI[7134] := 16#9B0F;
   // UNI[7135] := 16#9B13;
   // UNI[7136] := 16#9B1F;
   // UNI[7137] := 16#9B23;
   // UNI[7138] := 16#9B2F;
   // UNI[7139] := 16#9B32;
   // UNI[7140] := 16#9B3B;
   // UNI[7141] := 16#9B3C;
   // UNI[7142] := 16#9B41;
   // UNI[7143] := 16#9B42;
   // UNI[7144] := 16#9B43;
   // UNI[7145] := 16#9B44;
   // UNI[7146] := 16#9B45;
   // UNI[7147] := 16#9B47;
   // UNI[7148] := 16#9B48;
   // UNI[7149] := 16#9B49;
   // UNI[7150] := 16#9B4D;
   // UNI[7151] := 16#9B4F;
   // UNI[7152] := 16#9B51;
   // UNI[7153] := 16#9B54;
   // UNI[7154] := 16#9C7C;
   // UNI[7155] := 16#9C7F;
   // UNI[7156] := 16#9C81;
   // UNI[7157] := 16#9C82;
   // UNI[7158] := 16#9C85;
   // UNI[7159] := 16#9C86;
   // UNI[7160] := 16#9C87;
   // UNI[7161] := 16#9C88;
   // UNI[7162] := 16#9C8B;
   // UNI[7163] := 16#9C8D;
   // UNI[7164] := 16#9C8E;
   // UNI[7165] := 16#9C90;
   // UNI[7166] := 16#9C91;
